    PGN_AFTERTREATMENT_2_FUEL_CONTROL_2 : UDINT := UDINT#16#FD44; (* < 64836 - AT2FC2 *)
    PGN_AFTERTREATMENT_2_THREE_WAY_CATALYST : UDINT := UDINT#16#FD45; (* < 64837 - AT2TWC *)
    PGN_AFTERTREATMENT_1_THREE_WAY_CATALYST : UDINT := UDINT#16#FD46; (* < 64838 - AT1TWC *)
    PGN_TRANSMISSION_MODE_LABELS : UDINT := UDINT#16#FD47; (* < 64839 - TML *)
    PGN_ENGINE_EXHAUST_BANK_2_O2_FUEL_TRIM : UDINT := UDINT#16#FD48; (* < 64840 - O2FT2 *)
    PGN_ENGINE_EXHAUST_BANK_1_O2_FUEL_TRIM : UDINT := UDINT#16#FD49; (* < 64841 - O2FT1 *)
    PGN_GENERAL_PURPOSE_MESSAGE_2_11 : UDINT := UDINT#16#FD4A; (* < 64842 - GPM211 *)
    PGN_GENERAL_PURPOSE_MESSAGE_2_10 : UDINT := UDINT#16#FD4B; (* < 64843 - GPM210 *)
    PGN_GENERAL_PURPOSE_MESSAGE_2_9 : UDINT := UDINT#16#FD4C; (* < 64844 - GPM29 *)
    PGN_GENERAL_PURPOSE_MESSAGE_2_8 : UDINT := UDINT#16#FD4D; (* < 64845 - GPM28 *)
    PGN_GENERAL_PURPOSE_MESSAGE_2_7 : UDINT := UDINT#16#FD4E; (* < 64846 - GPM27 *)
    PGN_GENERAL_PURPOSE_MESSAGE_2_6 : UDINT := UDINT#16#FD4F; (* < 64847 - GPM26 *)
    PGN_GENERAL_PURPOSE_MESSAGE_1_9 : UDINT := UDINT#16#FD50; (* < 64848 - GPM19 *)
    PGN_AFTERCOOLER_COOLANT_CONTROL_VALVE_COMMAND : UDINT := UDINT#16#FD51; (* < 64849 - ACCVC *)
    PGN_ENGINE_COOLANT_CONTROL_VALVE_COMMAND : UDINT := UDINT#16#FD52; (* < 64850 - ECCVC *)
    PGN_ENGINE_AVERAGE_INFORMATION : UDINT := UDINT#16#FD53; (* < 64851 - EAI *)
    PGN_DTCS_C_PREVIOUSLY_ACTIVE : UDINT := UDINT#16#FD54; (* < 64852 - DM52 *)
    PGN_DTCS_C_CONFIRMED_AND_ACTIVE : UDINT := UDINT#16#FD55; (* < 64853 - DM51 *)
    PGN_DTCS_C_PENDING : UDINT := UDINT#16#FD56; (* < 64854 - DM50 *)
    PGN_DTCS_B2_PREVIOUSLY_ACTIVE : UDINT := UDINT#16#FD57; (* < 64855 - DM49 *)
    PGN_DTCS_B2_CONFIRMED_AND_ACTIVE : UDINT := UDINT#16#FD58; (* < 64856 - DM48 *)
    PGN_DTCS_B2_PENDING : UDINT := UDINT#16#FD59; (* < 64857 - DM47 *)
    PGN_DTCS_B1_PREVIOUSLY_ACTIVE : UDINT := UDINT#16#FD5A; (* < 64858 - DM46 *)
    PGN_DTCS_B1_CONFIRMED_AND_ACTIVE : UDINT := UDINT#16#FD5B; (* < 64859 - DM45 *)
    PGN_DTCS_B1_PENDING : UDINT := UDINT#16#FD5C; (* < 64860 - DM44 *)
    PGN_DTCS_A_PREVIOUSLY_ACTIVE : UDINT := UDINT#16#FD5D; (* < 64861 - DM43 *)
    PGN_DTCS_A_CONFIRMED_AND_ACTIVE : UDINT := UDINT#16#FD5E; (* < 64862 - DM42 *)
    PGN_DTCS_A_PENDING : UDINT := UDINT#16#FD5F; (* < 64863 - DM41 *)
    PGN_HARMONIZED_B1_FAILURE_COUNTS : UDINT := UDINT#16#FD60; (* < 64864 - DM40 *)
    PGN_HARMONIZED_CUMULATIVE_CONTINUOUS_MALFUNCTION_INDICATOR_SYSTEM : UDINT := UDINT#16#FD61; (* < 64865 - DM39 *)
    PGN_HARMONIZED_GLOBAL_REGULATION_DESCRIPTION : UDINT := UDINT#16#FD62; (* < 64866 - DM38 *)
    PGN_HARMONIZED_ROADWORTHINESS_SYSTEM : UDINT := UDINT#16#FD63; (* < 64867 - DM37 *)
    PGN_HARMONIZED_ROADWORTHINESS_VEHICLE : UDINT := UDINT#16#FD64; (* < 64868 - DM36 *)
    PGN_AFTERTREATMENT_1_FUEL_CONTROL_2 : UDINT := UDINT#16#FD65; (* < 64869 - AT1FC2 *)
    PGN_ENGINE_TEMPERATURE_4 : UDINT := UDINT#16#FD66; (* < 64870 - ET4 *)
    PGN_ZERO_NET_VEHICLE_WEIGHT_CHANGE : UDINT := UDINT#16#FD67; (* < 64871 - ZNVW *)
    PGN_GROSS_COMBINATION_VEHICLE_WEIGHT : UDINT := UDINT#16#FD68; (* < 64872 - GCVW *)
    PGN_AXLE_GROUP_CALIBRATION_WEIGHTS : UDINT := UDINT#16#FD69; (* < 64873 - AGCW *)
    PGN_AXLE_GROUP_WEIGHT : UDINT := UDINT#16#FD6A; (* < 64874 - AGW *)
    PGN_AVAILABLE_AXLE_GROUP_WEIGHTS : UDINT := UDINT#16#FD6B; (* < 64875 - AAGW *)
    PGN_AFTERTREATMENT_2_AIR_CONTROL_2 : UDINT := UDINT#16#FD6C; (* < 64876 - AT2AC2 *)
    PGN_AFTERTREATMENT_1_AIR_CONTROL_2 : UDINT := UDINT#16#FD6D; (* < 64877 - AT1AC2 *)
    PGN_AFTERTREATMENT_1_SCR_SERVICE_INFORMATION_1 : UDINT := UDINT#16#FD6E; (* < 64878 - A1SCRSI1 *)
    PGN_ELECTRONIC_ENGINE_CONTROLLER_8 : UDINT := UDINT#16#FD6F; (* < 64879 - EEC8 *)
    PGN_DOOR_RAMP_CONTROL : UDINT := UDINT#16#FD70; (* < 64880 - DRC *)
    PGN_BRAKE_ACTUATOR_STROKE_STATUS : UDINT := UDINT#16#FD71; (* < 64881 - BSA *)
    PGN_ENGINE_SPARK_VOLTAGE_6 : UDINT := UDINT#16#FD72; (* < 64882 - ESV6 *)
    PGN_ENGINE_SPARK_VOLTAGE_5 : UDINT := UDINT#16#FD73; (* < 64883 - ESV5 *)
    PGN_ENGINE_SPARK_VOLTAGE_4 : UDINT := UDINT#16#FD74; (* < 64884 - ESV4 *)
    PGN_ENGINE_SPARK_VOLTAGE_3 : UDINT := UDINT#16#FD75; (* < 64885 - ESV3 *)
    PGN_ENGINE_SPARK_VOLTAGE_2 : UDINT := UDINT#16#FD76; (* < 64886 - ESV2 *)
    PGN_ENGINE_SPARK_VOLTAGE_1 : UDINT := UDINT#16#FD77; (* < 64887 - ESV1 *)
    PGN_AFTERTREATMENT_2_TRIP_INFORMATION : UDINT := UDINT#16#FD78; (* < 64888 - AT2TI *)
    PGN_AFTERTREATMENT_1_TRIP_INFORMATION : UDINT := UDINT#16#FD79; (* < 64889 - AT1TI *)
    PGN_AFTERTREATMENT_2_SERVICE_1 : UDINT := UDINT#16#FD7A; (* < 64890 - AT2S1 *)
    PGN_AFTERTREATMENT_1_SERVICE_1 : UDINT := UDINT#16#FD7B; (* < 64891 - AT1S1 *)
    PGN_DIESEL_PARTICULATE_FILTER_CONTROL_1 : UDINT := UDINT#16#FD7C; (* < 64892 - DPFC1 *)
    PGN_RESERVED_FOR_FMS_TELLTALE_STATUS : UDINT := UDINT#16#FD7D; (* < 64893 - FMS1 *)
    PGN_ADAPTIVE_FRONT_LIGHTING_SYSTEM_STATUS : UDINT := UDINT#16#FD7E; (* < 64894 - AFSS *)
    PGN_ENGINE_CONFIGURATION_2 : UDINT := UDINT#16#FD7F; (* < 64895 - EC2 *)
    PGN_EMISSION_RELATED_PERMANENT_DIAGNOSTIC_TROUBLE_CODES : UDINT := UDINT#16#FD80; (* < 64896 - DM28 *)
    PGN_EGR_COOLER_BYPASS : UDINT := UDINT#16#FD81; (* < 64897 - EGRBV *)
    PGN_ALL_PENDING_DTCS : UDINT := UDINT#16#FD82; (* < 64898 - DM27 *)
    PGN_TRANSFER_CASE_INFORMATION : UDINT := UDINT#16#FD83; (* < 64899 - TCI *)
    PGN_ENGINE_FLUID_LEVEL_PRESSURE_9 : UDINT := UDINT#16#FD84; (* < 64900 - EFL/P9 *)
    PGN_ENGINE_FLUID_LEVEL_PRESSURE_8 : UDINT := UDINT#16#FD85; (* < 64901 - EFL/P8 *)
    PGN_ENGINE_FLUID_LEVEL_PRESSURE_7 : UDINT := UDINT#16#FD86; (* < 64902 - EFL/P7 *)
    PGN_ENGINE_FLUID_LEVEL_PRESSURE_6 : UDINT := UDINT#16#FD87; (* < 64903 - EFL/P6 *)
    PGN_ENGINE_FLUID_LEVEL_PRESSURE_5 : UDINT := UDINT#16#FD88; (* < 64904 - EFL/P5 *)
    PGN_VEHICLE_DIRECTION_SPEED_2 : UDINT := UDINT#16#FD89; (* < 64905 - VDS2 *)
    PGN_SAE_J2012_2_BYTE_DTC_DISPLAY : UDINT := UDINT#16#FD8A; (* < 64906 - J2012_2B *)
    PGN_AFTERTREATMENT_2_GAS_PARAMETERS : UDINT := UDINT#16#FD8B; (* < 64907 - AT2GP *)
    PGN_AFTERTREATMENT_1_GAS_PARAMETERS : UDINT := UDINT#16#FD8C; (* < 64908 - AT1GP *)
    PGN_UTILITY_TOTAL_AC_REACTIVE_ENERGY : UDINT := UDINT#16#FD8D; (* < 64909 - UTACER *)
    PGN_GENERATOR_TOTAL_AC_REACTIVE_ENERGY : UDINT := UDINT#16#FD8E; (* < 64910 - GTACER *)
    PGN_GENERATOR_TOTAL_AC_PERCENT_POWER : UDINT := UDINT#16#FD8F; (* < 64911 - GTACPP *)
    PGN_ADVERTISED_ENGINE_TORQUE_CURVE : UDINT := UDINT#16#FD90; (* < 64912 - AETC *)
    PGN_AC_SWITCHING_DEVICE_STATUS : UDINT := UDINT#16#FD91; (* < 64913 - ACS *)
    PGN_ENGINE_OPERATING_INFORMATIO : UDINT := UDINT#16#FD92; (* < 64914 - EOI *)
    PGN_GENERATOR_CONTROL_1 : UDINT := UDINT#16#FD93; (* < 64915 - GC1 *)
    PGN_ELECTRONIC_ENGINE_CONTROLLER_7 : UDINT := UDINT#16#FD94; (* < 64916 - EEC7 *)
    PGN_TRANSMISSION_FLUIDS_2 : UDINT := UDINT#16#FD95; (* < 64917 - TRF2 *)
    PGN_FUEL_INFORMATION_2_LIQUID : UDINT := UDINT#16#FD96; (* < 64918 - LFI2 *)
    PGN_FUEL_INFORMATION_3_LIQUID : UDINT := UDINT#16#FD97; (* < 64919 - LFI3 *)
    PGN_AFTERTREATMENT_1_HISTORICAL_INFORMATION_1 : UDINT := UDINT#16#FD98; (* < 64920 - AT1HI1 *)
    PGN_AFTERTREATMENT_2_HISTORICAL_INFORMATION_1 : UDINT := UDINT#16#FD99; (* < 64921 - AT2HI1 *)
    PGN_ELECTRONIC_BRAKE_SYSTEM_2_4 : UDINT := UDINT#16#FD9A; (* < 64922 - EBS24 *)
    PGN_AFTERTREATMENT_1_DIESEL_EXHAUST_FLUID_INFORMATION_1 : UDINT := UDINT#16#FD9B; (* < 64923 - A1DEFI1 *)
    PGN_SENSOR_ELECTRICAL_POWER_2 : UDINT := UDINT#16#FD9C; (* < 64924 - SEP2 *)
    PGN_SENSOR_ELECTRICAL_POWER_1 : UDINT := UDINT#16#FD9D; (* < 64925 - SEP1 *)
    PGN_AFTERTREATMENT_2_AIR_CONTROL_1 : UDINT := UDINT#16#FD9E; (* < 64926 - AT2AC1 *)
    PGN_AFTERTREATMENT_1_AIR_CONTROL_1 : UDINT := UDINT#16#FD9F; (* < 64927 - AT1AC1 *)
    PGN_AFTERTREATMENT_2_FUEL_CONTROL_1 : UDINT := UDINT#16#FDA0; (* < 64928 - AT2FC1 *)
    PGN_AFTERTREATMENT_1_FUEL_CONTROL_1 : UDINT := UDINT#16#FDA1; (* < 64929 - AT1FC1 *)
    PGN_FUEL_INFORMATION_3_GASEOUS : UDINT := UDINT#16#FDA2; (* < 64930 - GFI3 *)
    PGN_ELECTRONIC_ENGINE_CONTROLLER_6 : UDINT := UDINT#16#FDA3; (* < 64931 - EEC6 *)
    PGN_PTO_DRIVE_ENGAGEMENT_1 : UDINT := UDINT#16#FDA4; (* < 64932 - PTODE1 *)
    PGN_DOOR_CONTROL_2 : UDINT := UDINT#16#FDA5; (* < 64933 - DC2 *)
    PGN_VOLTAGE_REGULATOR_EXCITATION_STATUS : UDINT := UDINT#16#FDA6; (* < 64934 - VREP *)
    PGN_VOLTAGE_REGULATOR_OPERATING_MODE : UDINT := UDINT#16#FDA7; (* < 64935 - VROM *)
    PGN_WIRELESS_COMMUNICATIONS_MESSAGE_2 : UDINT := UDINT#16#FDA8; (* < 64936 - WCM2 *)
    PGN_WCM1 : UDINT := UDINT#16#FDA9; (* < 64937 - WCM1 *)
    PGN_ENGINE_FLUID_LEVEL_PRESSURE_4 : UDINT := UDINT#16#FDAA; (* < 64938 - EFL/P4 *)
    PGN_REQUEST_FOR_COMPLETE_CONFIGURABLE_MESSAGE_SET_NO_LONGER_USED : UDINT := UDINT#16#FDAB; (* < 64939 - Request For Complete Configurable Message Set (no longer used) *)
    PGN_ENGINE_FUEL_INFORMATION : UDINT := UDINT#16#FDAC; (* < 64940 - EFI *)
    PGN_REQUEST_FOR_COMPLETE_CONFIGURABLE_MESSAGE_SET : UDINT := UDINT#16#FDAD; (* < 64941 - RCMS *)
    PGN_FIFTH_WHEEL_SMART_SYSTEMS_2 : UDINT := UDINT#16#FDAE; (* < 64942 - FWSS2 *)
    PGN_AFTERTREATMENT_2_INTERMEDIATE_GAS : UDINT := UDINT#16#FDAF; (* < 64943 - AT2IMG *)
    PGN_AFTERTREATMENT_2_OUTLET_GAS_2 : UDINT := UDINT#16#FDB0; (* < 64944 - AT2OG2 *)
    PGN_AFTERTREATMENT_2_INTAKE_GAS_2 : UDINT := UDINT#16#FDB1; (* < 64945 - AT2IG2 *)
    PGN_AFTERTREATMENT_1_INTERMEDIATE_GAS : UDINT := UDINT#16#FDB2; (* < 64946 - AT1IMG *)
    PGN_AFTERTREATMENT_1_OUTLET_GAS_2 : UDINT := UDINT#16#FDB3; (* < 64947 - AT1OG2 *)
    PGN_AFTERTREATMENT_1_INTAKE_GAS_2 : UDINT := UDINT#16#FDB4; (* < 64948 - AT1IG2 *)
    PGN_EMISSION_RELATED_PREVIOUSLY_MIL_ON_DIAGNOSTIC_TROUBLE_CODES : UDINT := UDINT#16#FDB5; (* < 64949 - DM23 *)
    PGN_SPN_SUPPORT : UDINT := UDINT#16#FDB6; (* < 64950 - DM24 *)
    PGN_EXPANDED_FREEZE_FRAME : UDINT := UDINT#16#FDB7; (* < 64951 - DM25 *)
    PGN_DIAGNOSTIC_READINESS_3 : UDINT := UDINT#16#FDB8; (* < 64952 - DM26 *)
    PGN_TIRE_PRESSURE_REFERENCE_INFORMATION : UDINT := UDINT#16#FDB9; (* < 64953 - TPRI *)
    PGN_FAREBOX_STATUS : UDINT := UDINT#16#FDBA; (* < 64954 - TR6 *)
    PGN_FAREBOX_POINT_OF_SALE : UDINT := UDINT#16#FDBB; (* < 64955 - TR5 *)
    PGN_FAREBOX_SERVICE_DETAIL : UDINT := UDINT#16#FDBC; (* < 64956 - TR4 *)
    PGN_SIGNAL_PREEMPTION : UDINT := UDINT#16#FDBD; (* < 64957 - TR3 *)
    PGN_TRANSIT_ROUTE : UDINT := UDINT#16#FDBE; (* < 64958 - TR1 *)
    PGN_TRANSIT_MILEPOST : UDINT := UDINT#16#FDBF; (* < 64959 - TR2 *)
    PGN_PASSENGER_COUNTER : UDINT := UDINT#16#FDC0; (* < 64960 - TR7 *)
    PGN_ENGINE_FLUID_LEVEL_PRESSURE_3 : UDINT := UDINT#16#FDC1; (* < 64961 - EFL/P3 *)
    PGN_ELECTRONIC_ENGINE_CONTROLLER_14 : UDINT := UDINT#16#FDC2; (* < 64962 - EEC14 *)
    PGN_ELECTRONIC_ENGINE_CONTROLLER_15 : UDINT := UDINT#16#FDC3; (* < 64963 - EEC15 *)
    PGN_ELECTRONIC_BRAKE_CONTROLLER_5 : UDINT := UDINT#16#FDC4; (* < 64964 - EBC5 *)
    PGN_ECU_IDENTIFICATION_INFO : UDINT := UDINT#16#FDC5; (* < 64965 - ECUID *)
    PGN_COLD_START_AIDS : UDINT := UDINT#16#FDC6; (* < 64966 - CSA *)
    PGN_OFF_HIGHWAY_ENGINE_CONTROL_SELECTION_STATES : UDINT := UDINT#16#FDC7; (* < 64967 - OHCSS *)
    PGN_OPERATOR_PRIMARY_INTERMEDIATE_SPEED_CONTROL_STATE : UDINT := UDINT#16#FDC8; (* < 64968 - ISCS *)
    PGN_ELECTRONIC_CONTROL_MODULE_INFORMATION : UDINT := UDINT#16#FDC9; (* < 64969 - CMI *)
    PGN_INTERMEDIATE_SPEED_CONTROL : UDINT := UDINT#16#FDCA; (* < 64970 - ISC *)
    PGN_OFFHIGHW_ENGINE_CTRL_SELECT : UDINT := UDINT#16#FDCB; (* < 64971 - OHECS *)
    PGN_OPERATORS_EXTERNAL_LIGHT_CONTROLS_MESSAGE : UDINT := UDINT#16#FDCC; (* < 64972 - OEL *)
    PGN_OPERATOR_WIPER_AND_WASHER_CONTROLS_MESSAGE : UDINT := UDINT#16#FDCD; (* < 64973 - OWW *)
    PGN_WORKING_SET_MEMBER_MESSAGE_OBSOLETE_SEE_PGN_65088 : UDINT := UDINT#16#FDCE; (* < 64974 - WSMM *)
    PGN_WORKING_SET_MASTER_MESSAGE_OBSOLETE_SEE_PGN_65089 : UDINT := UDINT#16#FDCF; (* < 64975 - WSM *)
    PGN_INTAKE_EXHAUST_CONDITIONS_2 : UDINT := UDINT#16#FDD0; (* < 64976 - IC2 *)
    PGN_FMS_STANDARD_INTERFAC_IDENT : UDINT := UDINT#16#FDD1; (* < 64977 - FMS *)
    PGN_ECU_PERFORMANCE : UDINT := UDINT#16#FDD2; (* < 64978 - EP *)
    PGN_TURBOCHARGER_INFORMATION_6 : UDINT := UDINT#16#FDD3; (* < 64979 - TCI6 *)
    PGN_CAB_MESSAGE_3 : UDINT := UDINT#16#FDD4; (* < 64980 - CM3 *)
    PGN_ELEC_ENGINE_CONTROLLER_5 : UDINT := UDINT#16#FDD5; (* < 64981 - EEC5 *)
    PGN_BASIC_JOYSTICK_MESSAGE_1 : UDINT := UDINT#16#FDD6; (* < 64982 - BJM1 *)
    PGN_EXTENDED_JOYSTICK_MESSAGE_1 : UDINT := UDINT#16#FDD7; (* < 64983 - EJM1 *)
    PGN_BASIC_JOYSTICK_MESSAGE_2 : UDINT := UDINT#16#FDD8; (* < 64984 - BJM2 *)
    PGN_EXTENDED_JOYSTICK_MESSAGE_2 : UDINT := UDINT#16#FDD9; (* < 64985 - EJM2 *)
    PGN_BASIC_JOYSTICK_MESSAGE_3 : UDINT := UDINT#16#FDDA; (* < 64986 - BJM3 *)
    PGN_EXTENDED_JOYSTICK_MESSAGE_3 : UDINT := UDINT#16#FDDB; (* < 64987 - EJM3 *)
    PGN_MARINE_CONTROL_INFORMATION : UDINT := UDINT#16#FDDC; (* < 64988 - MCI *)
    PGN_MILITARY_APPLICATION_MESSAGE_1_1 : UDINT := UDINT#16#FDDD; (* < 64989 - MAM11 *)
    PGN_AMBIENT_CONDITIONS_2 : UDINT := UDINT#16#FDDE; (* < 64990 - MAM21 *)
    PGN_FRONT_WHEEL_DRIVE_STATUS : UDINT := UDINT#16#FDDF; (* < 64991 - FWD *)
    PGN_AMBIENT_CONDITIONS_2_64992 : UDINT := UDINT#16#FDE0; (* < 64992 - AMB2 *)
    PGN_CAB_A_C_CLIMATE_SYST_INFO : UDINT := UDINT#16#FDE1; (* < 64993 - CCSI1 *)
    PGN_SUPPLY_PRESSURE_DEMAND : UDINT := UDINT#16#FDE2; (* < 64994 - SPR *)
    PGN_EQUIPM_OPERATION_AND_CONTR : UDINT := UDINT#16#FDE3; (* < 64995 - EOAC *)
    PGN_EQUIPMENT_PERFORMANCE_DATA : UDINT := UDINT#16#FDE4; (* < 64996 - EPD *)
    PGN_MAX_VEHIC_SPEED_LIMIT_STAT : UDINT := UDINT#16#FDE5; (* < 64997 - MVS *)
    PGN_HYDRAULIC_BRAKING_SYSTEM : UDINT := UDINT#16#FDE6; (* < 64998 - HBS *)
    PGN_BUS_1_UTIL_SYNC_CHECK_STATU : UDINT := UDINT#16#FDE7; (* < 64999 - BUSC *)
    PGN_BUS_1_GENERA_SYNC_CH_STAT : UDINT := UDINT#16#FDE8; (* < 65000 - BGSC *)
    PGN_BUS_1_PHASE_C_BASIC_AC_QUAN : UDINT := UDINT#16#FDE9; (* < 65001 - BPCAC *)
    PGN_BUS_1_PHASE_B_BASIC_AC_QUAN : UDINT := UDINT#16#FDEA; (* < 65002 - BPBAC *)
    PGN_BUS_1_PHASE_A_BASIC_AC_QUAN : UDINT := UDINT#16#FDEB; (* < 65003 - BPAAC *)
    PGN_BUS_1_AVERAGE_BASIC_AC_QUAN : UDINT := UDINT#16#FDEC; (* < 65004 - BAAC *)
    PGN_UTIL_TOTAL_AC_ENERGY : UDINT := UDINT#16#FDED; (* < 65005 - UTACE *)
    PGN_UTIL_PHASE_C_AC_REACT_POWER : UDINT := UDINT#16#FDEE; (* < 65006 - UPCACR *)
    PGN_UTIL_PHASE_C_AC_POWER : UDINT := UDINT#16#FDEF; (* < 65007 - UPCACP *)
    PGN_UTIL_PHASE_C_AC_BASIC_QUANT : UDINT := UDINT#16#FDF0; (* < 65008 - UPCAC *)
    PGN_UTIL_PHASE_B_AC_REACT_POWER : UDINT := UDINT#16#FDF1; (* < 65009 - UPBACR *)
    PGN_UTIL_PHASE_B_AC_POWER : UDINT := UDINT#16#FDF2; (* < 65010 - UPBACP *)
    PGN_UTIL_PHASE_B_AC_BASIC_QUANT : UDINT := UDINT#16#FDF3; (* < 65011 - UPBAC *)
    PGN_UTIL_PHASE_A_AC_REACT_POWER : UDINT := UDINT#16#FDF4; (* < 65012 - UPACCR *)
    PGN_UTIL_PHASE_A_AC_POWER : UDINT := UDINT#16#FDF5; (* < 65013 - UPAACP *)
    PGN_UTIL_PHASE_A_AC_BASIC_QUANT : UDINT := UDINT#16#FDF6; (* < 65014 - UPAAC *)
    PGN_UTIL_AC_REACTIVE_POWER : UDINT := UDINT#16#FDF7; (* < 65015 - UTACR *)
    PGN_UTIL_TOTAL_AC_POWER : UDINT := UDINT#16#FDF8; (* < 65016 - UTACP *)
    PGN_UTIL_AVERACE_BASIC_AC_QUANT : UDINT := UDINT#16#FDF9; (* < 65017 - UAAC *)
    PGN_GENERATOR_TOTAL_AC_ENERGY : UDINT := UDINT#16#FDFA; (* < 65018 - GTACE *)
    PGN_GENERA_PHAS_C_AC_REACT_PWR : UDINT := UDINT#16#FDFB; (* < 65019 - GPCACR *)
    PGN_GENERATOR_PHASE_C_AC_POWER : UDINT := UDINT#16#FDFC; (* < 65020 - GPCACP *)
    PGN_GENERA_PHASE_C_BAS_AC_QUANT : UDINT := UDINT#16#FDFD; (* < 65021 - GPCAC *)
    PGN_GENERA_PHASE_B_AC_REACT_PWR : UDINT := UDINT#16#FDFE; (* < 65022 - GPBACRP *)
    PGN_GENERATOR_PHASE_B_AC_POWER : UDINT := UDINT#16#FDFF; (* < 65023 - GPBACP *)
    PGN_PDU2_254_Y : UDINT := UDINT#16#FE00; (* < 65024 - GPBAC *)
    PGN_GENERA_PHASE_B_BAS_AC_QUANT : UDINT := UDINT#16#FE00; (* < 65024 - GPBAC *)
    PGN_GENERA_PHASE_A_AC_REACT_PWR : UDINT := UDINT#16#FE01; (* < 65025 - GPAACR *)
    PGN_GENERATOR_PHASE_A_AC_POWER : UDINT := UDINT#16#FE02; (* < 65026 - GPAACP *)
    PGN_GENERA_PHASE_A_BAS_AC_QUANT : UDINT := UDINT#16#FE03; (* < 65027 - GPAAC *)
    PGN_GENERA_TOTAL_AC_REACT_POWER : UDINT := UDINT#16#FE04; (* < 65028 - GTACR *)
    PGN_GENERATOR_TOTAL_AC_POWER : UDINT := UDINT#16#FE05; (* < 65029 - GTACP *)
    PGN_GENERA_TOTAL_BAS_AC_QUANTI : UDINT := UDINT#16#FE06; (* < 65030 - GAAC *)
    PGN_EXHAUST_TEMPERATURE : UDINT := UDINT#16#FE07; (* < 65031 - ET *)
    PGN_REQUIRED_TRACTOR_FACILITIES : UDINT := UDINT#16#FE08; (* < 65032 - RTF *)
    PGN_TRACTOR_FACILITIES_RESPONSE : UDINT := UDINT#16#FE09; (* < 65033 - TFR *)
    PGN_IMP_REMOTE_CMD_TRACTOR_RESP : UDINT := UDINT#16#FE0A; (* < 65034 - IRCR *)
    PGN_IMPLEMENT_REMOTE_CONTR_CMD : UDINT := UDINT#16#FE0B; (* < 65035 - IRC *)
    PGN_WORKING_SET_MEMBER : UDINT := UDINT#16#FE0C; (* < 65036 - WSMEM *)
    PGN_WORKING_SET_MASTER : UDINT := UDINT#16#FE0D; (* < 65037 - WSMSTR *)
    PGN_RESP_FOR_REPETITION_RATE : UDINT := UDINT#16#FE0E; (* < 65038 - RESRR *)
    PGN_LANGUAGE_COMMAND : UDINT := UDINT#16#FE0F; (* < 65039 - LC *)
    PGN_AUX_VALVE_0_EST_FLOW : UDINT := UDINT#16#FE10; (* < 65040 - AV00EF *)
    PGN_AUX_VALVE_1_EST_FLOW : UDINT := UDINT#16#FE11; (* < 65041 - AV01EF *)
    PGN_AUX_VALVE_2_EST_FLOW : UDINT := UDINT#16#FE12; (* < 65042 - AV02EF *)
    PGN_AUX_VALVE_3_EST_FLOW : UDINT := UDINT#16#FE13; (* < 65043 - AV03EF *)
    PGN_AUX_VALVE_4_EST_FLOW : UDINT := UDINT#16#FE14; (* < 65044 - AV04EF *)
    PGN_AUX_VALVE_5_EST_FLOW : UDINT := UDINT#16#FE15; (* < 65045 - AV05EF *)
    PGN_AUX_VALVE_6_EST_FLOW : UDINT := UDINT#16#FE16; (* < 65046 - AV06EF *)
    PGN_AUX_VALVE_7_EST_FLOW : UDINT := UDINT#16#FE17; (* < 65047 - AV07EF *)
    PGN_AUX_VALVE_8_EST_FLOW : UDINT := UDINT#16#FE18; (* < 65048 - AV08EF *)
    PGN_AUX_VALVE_9_EST_FLOW : UDINT := UDINT#16#FE19; (* < 65049 - AV09EF *)
    PGN_AUX_VALVE_10_EST_FLOW : UDINT := UDINT#16#FE1A; (* < 65050 - AV10EF *)
    PGN_AUX_VALVE_11_EST_FLOW : UDINT := UDINT#16#FE1B; (* < 65051 - AV11EF *)
    PGN_AUX_VALVE_12_EST_FLOW : UDINT := UDINT#16#FE1C; (* < 65052 - AV12EF *)
    PGN_AUX_VALVE_13_EST_FLOW : UDINT := UDINT#16#FE1D; (* < 65053 - AV13EF *)
    PGN_AUX_VALVE_14_EST_FLOW : UDINT := UDINT#16#FE1E; (* < 65054 - AV14EF *)
    PGN_AUX_VALVE_15_EST_FLOW : UDINT := UDINT#16#FE1F; (* < 65055 - AV15EF *)
    PGN_AUX_VALVE_0_MEAS_FLOW : UDINT := UDINT#16#FE20; (* < 65056 - AV00MF *)
    PGN_AUX_VALVE_1_MEAS_FLOW : UDINT := UDINT#16#FE21; (* < 65057 - AV01MF *)
    PGN_AUX_VALVE_2_MEAS_FLOW : UDINT := UDINT#16#FE22; (* < 65058 - AV02MF *)
    PGN_AUX_VALVE_3_MEAS_FLOW : UDINT := UDINT#16#FE23; (* < 65059 - AV03MF *)
    PGN_AUX_VALVE_4_MEAS_FLOW : UDINT := UDINT#16#FE24; (* < 65060 - AV04MF *)
    PGN_AUX_VALVE_5_MEAS_FLOW : UDINT := UDINT#16#FE25; (* < 65061 - AV05MF *)
    PGN_AUX_VALVE_6_MEAS_FLOW : UDINT := UDINT#16#FE26; (* < 65062 - AV06MF *)
    PGN_AUX_VALVE_7_MEAS_FLOW : UDINT := UDINT#16#FE27; (* < 65063 - AV07MF *)
    PGN_AUX_VALVE_8_MEAS_FLOW : UDINT := UDINT#16#FE28; (* < 65064 - AV08MF *)
    PGN_AUX_VALVE_9_MEAS_FLOW : UDINT := UDINT#16#FE29; (* < 65065 - AV09MF *)
    PGN_AUX_VALVE_10_MEAS_FLOW : UDINT := UDINT#16#FE2A; (* < 65066 - AV10MF *)
    PGN_AUX_VALVE_11_MEAS_FLOW : UDINT := UDINT#16#FE2B; (* < 65067 - AV11MF *)
    PGN_AUX_VALVE_12_MEAS_FLOW : UDINT := UDINT#16#FE2C; (* < 65068 - AV12MF *)
    PGN_AUX_VALVE_13_MEAS_FLOW : UDINT := UDINT#16#FE2D; (* < 65069 - AV13MF *)
    PGN_AUX_VALVE_14_MEAS_FLOW : UDINT := UDINT#16#FE2E; (* < 65070 - AV14MF *)
    PGN_AUX_VALVE_15_MEAS_FLOW : UDINT := UDINT#16#FE2F; (* < 65071 - AV15MF *)
    PGN_AUX_VALVE_0_COMMAND : UDINT := UDINT#16#FE30; (* < 65072 - AV00C *)
    PGN_AUX_VALVE_1_COMMAND : UDINT := UDINT#16#FE31; (* < 65073 - AV01C *)
    PGN_AUX_VALVE_2_COMMAND : UDINT := UDINT#16#FE32; (* < 65074 - AV02C *)
    PGN_AUX_VALVE_3_COMMAND : UDINT := UDINT#16#FE33; (* < 65075 - AV03C *)
    PGN_AUX_VALVE_4_COMMAND : UDINT := UDINT#16#FE34; (* < 65076 - AV04C *)
    PGN_AUX_VALVE_5_COMMAND : UDINT := UDINT#16#FE35; (* < 65077 - AV05C *)
    PGN_AUX_VALVE_6_COMMAND : UDINT := UDINT#16#FE36; (* < 65078 - AV06C *)
    PGN_AUX_VALVE_7_COMMAND : UDINT := UDINT#16#FE37; (* < 65079 - AV07C *)
    PGN_AUX_VALVE_8_COMMAND : UDINT := UDINT#16#FE38; (* < 65080 - AV08C *)
    PGN_AUX_VALVE_9_COMMAND : UDINT := UDINT#16#FE39; (* < 65081 - AV09C *)
    PGN_AUX_VALVE_10_COMMAND : UDINT := UDINT#16#FE3A; (* < 65082 - AV10C *)
    PGN_AUX_VALVE_11_COMMAND : UDINT := UDINT#16#FE3B; (* < 65083 - AV11C *)
    PGN_AUX_VALVE_12_COMMAND : UDINT := UDINT#16#FE3C; (* < 65084 - AV12C *)
    PGN_AUX_VALVE_13_COMMAND : UDINT := UDINT#16#FE3D; (* < 65085 - AV13C *)
    PGN_AUX_VALVE_14_COMMAND : UDINT := UDINT#16#FE3E; (* < 65086 - AV14C *)
    PGN_AUX_VALVE_15_COMMAND : UDINT := UDINT#16#FE3F; (* < 65087 - AV15C *)
    PGN_LIGHTING_DATA : UDINT := UDINT#16#FE40; (* < 65088 - LD *)
    PGN_LIGHTING_COMMAND : UDINT := UDINT#16#FE41; (* < 65089 - LCMD *)
    PGN_COMMAND_HITCH_PTO : UDINT := UDINT#16#FE42; (* < 65090 - HPTOC *)
    PGN_REAR_PTO : UDINT := UDINT#16#FE43; (* < 65091 - RPTO *)
    PGN_FRONT_PTO : UDINT := UDINT#16#FE44; (* < 65092 - FPTO *)
    PGN_REAR_HITCH : UDINT := UDINT#16#FE45; (* < 65093 - RHS *)
    PGN_FRONT_HITCH : UDINT := UDINT#16#FE46; (* < 65094 - FHS *)
    PGN_MAINTAIN_POWER : UDINT := UDINT#16#FE47; (* < 65095 - MP *)
    PGN_WHEEL_BASED_SPEED : UDINT := UDINT#16#FE48; (* < 65096 - WBSD *)
    PGN_GROUND_BASED_SPEED : UDINT := UDINT#16#FE49; (* < 65097 - GBSD *)
    PGN_ELECTRONIC_TRANSMISSION_CONTROLLER_7 : UDINT := UDINT#16#FE4A; (* < 65098 - ETC7 *)
    PGN_TRANSMISSIONG_CONFIG_2 : UDINT := UDINT#16#FE4B; (* < 65099 - TCFG2 *)
    PGN_MILITARY_LIGHTING_COMMAND : UDINT := UDINT#16#FE4C; (* < 65100 - ML *)
    PGN_TOTAL_AVERAGED_INFORMATION : UDINT := UDINT#16#FE4D; (* < 65101 - TAVG *)
    PGN_DOOR_CONTROL : UDINT := UDINT#16#FE4E; (* < 65102 - DC1 *)
    PGN_VEHICLE_DYN_STAB_CTRL_1 : UDINT := UDINT#16#FE4F; (* < 65103 - VDC1 *)
    PGN_BATTERY_TEMPERATURE : UDINT := UDINT#16#FE50; (* < 65104 - BT1 *)
    PGN_ADAPT_CRUISE_CONTR_OPER_INP : UDINT := UDINT#16#FE51; (* < 65105 - ACC2 *)
    PGN_VEHICLE_ELECTRICAL_POWER_3 : UDINT := UDINT#16#FE52; (* < 65106 - VEP3 *)
    PGN_RETARD_TORQUE_SPEED_LIMIT : UDINT := UDINT#16#FE53; (* < 65107 - RTC1 *)
    PGN_ENGINE_TORQUE_SPEED_LIMIT : UDINT := UDINT#16#FE54; (* < 65108 - ECT1 *)
    PGN_GASEOUS_FUEL_PROPERTIES : UDINT := UDINT#16#FE55; (* < 65109 - GFD *)
    PGN_TANK_INFORMATION_1 : UDINT := UDINT#16#FE56; (* < 65110 - AT1T1I1 *)
    PGN_AIR_SUSPENSION_CONTROL_5 : UDINT := UDINT#16#FE57; (* < 65111 - ASC5 *)
    PGN_AIR_SUSPENSION_CONTROL_4 : UDINT := UDINT#16#FE58; (* < 65112 - ASC4 *)
    PGN_AIR_SUSPENSION_CONTROL_3 : UDINT := UDINT#16#FE59; (* < 65113 - ASC3 *)
    PGN_AIR_SUSPENSION_CONTROL_1 : UDINT := UDINT#16#FE5A; (* < 65114 - ASC1 *)
    PGN_FORWARD_LANE_IMAGE : UDINT := UDINT#16#FE5B; (* < 65115 - FLI2 *)
    PGN_RUNNING_GEAR_EQUIPMENT_2_2 : UDINT := UDINT#16#FE5C; (* < 65116 - RGE22 *)
    PGN_GENERAL_PURPOSE_MESSAGE_1_2 : UDINT := UDINT#16#FE5D; (* < 65117 - GPM12 *)
    PGN_RUNNING_GEAR_EQUIPMENT_2_3 : UDINT := UDINT#16#FE5E; (* < 65118 - RGE23 *)
    PGN_GENERAL_PURPOSE_MESSAGE_1_3 : UDINT := UDINT#16#FE5F; (* < 65119 - GPM13 *)
    PGN_GENERAL_PURPOSE_MESSAGE_2_3 : UDINT := UDINT#16#FE60; (* < 65120 - GPM23 *)
    PGN_GENERAL_PURPOSE_MESSAGE_1_4 : UDINT := UDINT#16#FE61; (* < 65121 - GPM14 *)
    PGN_GENERAL_PURPOSE_MESSAGE_2_4 : UDINT := UDINT#16#FE62; (* < 65122 - GPM24 *)
    PGN_GENERAL_PURPOSE_MESSAGE_1_5 : UDINT := UDINT#16#FE63; (* < 65123 - GPM15 *)
    PGN_GENERAL_PURPOSE_MESSAGE_2_5 : UDINT := UDINT#16#FE64; (* < 65124 - GPM25 *)
    PGN_GENERAL_PURPOSE_MESSAGE_1_6 : UDINT := UDINT#16#FE65; (* < 65125 - GPM16 *)
    PGN_BATTERY_MAIN_SWITCH_INFO : UDINT := UDINT#16#FE66; (* < 65126 - BM *)
    PGN_CLIMATE_CONTR_CONFIGURATION : UDINT := UDINT#16#FE67; (* < 65127 - CCC *)
    PGN_VEHICLE_FLUIDS : UDINT := UDINT#16#FE68; (* < 65128 - VF *)
    PGN_ENGINE_TEMPERATURE_3 : UDINT := UDINT#16#FE69; (* < 65129 - ET3 *)
    PGN_ENGINE_FUEL_LUBE_SYSTEMS : UDINT := UDINT#16#FE6A; (* < 65130 - EFS *)
    PGN_DRIVERS_IDENTIFICATION : UDINT := UDINT#16#FE6B; (* < 65131 - DI *)
    PGN_TACHOGRAPH : UDINT := UDINT#16#FE6C; (* < 65132 - TCO1 *)
    PGN_HEATER_INFORMATION : UDINT := UDINT#16#FE6D; (* < 65133 - HTR *)
    PGN_HIGH_RESOLUTION_WHEEL_SPEED : UDINT := UDINT#16#FE6E; (* < 65134 - HRW *)
    PGN_ADAPTIVE_CRUISE_CONTROL : UDINT := UDINT#16#FE6F; (* < 65135 - ACC1 *)
    PGN_COMBINATION_VEHICLE_WEIGHT : UDINT := UDINT#16#FE70; (* < 65136 - CVW *)
    PGN_LASER_TRACER_POSITION : UDINT := UDINT#16#FE71; (* < 65137 - LTP *)
    PGN_LASER_LEVEL_SYS_BLADE_CONTR : UDINT := UDINT#16#FE72; (* < 65138 - LBC *)
    PGN_LASER_RECEIVER_MAST_POS : UDINT := UDINT#16#FE73; (* < 65139 - LMP *)
    PGN_MODIFY_LEVEL_CTRL_SET_POINT : UDINT := UDINT#16#FE74; (* < 65140 - LSP *)
    PGN_LASER_LVL_SYS_VERTIC_DEVIAT : UDINT := UDINT#16#FE75; (* < 65141 - LVD *)
    PGN_LASER_LVL_SYS_POS_DISP_DATA : UDINT := UDINT#16#FE76; (* < 65142 - LVDD *)
    PGN_AUXILIARY_PRESSURES : UDINT := UDINT#16#FE77; (* < 65143 - AP *)
    PGN_TIRE_PRESS_CONTR_UNIT_STAT : UDINT := UDINT#16#FE78; (* < 65144 - TP1 *)
    PGN_TIRE_PRESS_CTRL_TARGET_PRES : UDINT := UDINT#16#FE79; (* < 65145 - TP2 *)
    PGN_TIRE_PRESS_UNIT_CURR_PRESS : UDINT := UDINT#16#FE7A; (* < 65146 - TP3 *)
    PGN_COMBUSTION_TIME_1 : UDINT := UDINT#16#FE7B; (* < 65147 - CT1 *)
    PGN_COMBUSTION_TIME_2 : UDINT := UDINT#16#FE7C; (* < 65148 - CT2 *)
    PGN_COMBUSTION_TIME_3 : UDINT := UDINT#16#FE7D; (* < 65149 - CT3 *)
    PGN_COMBUSTION_TIME_4 : UDINT := UDINT#16#FE7E; (* < 65150 - CT4 *)
    PGN_COMBUSTION_TIME_5 : UDINT := UDINT#16#FE7F; (* < 65151 - CT5 *)
    PGN_COMBUSTION_TIME_6 : UDINT := UDINT#16#FE80; (* < 65152 - CT6 *)
    PGN_FUEL_INFORMATION_2 : UDINT := UDINT#16#FE81; (* < 65153 - GFI2 *)
    PGN_IGNITION_TIMING_1 : UDINT := UDINT#16#FE82; (* < 65154 - IT1 *)
    PGN_IGNITION_TIMING_2 : UDINT := UDINT#16#FE83; (* < 65155 - IT2 *)
    PGN_IGNITION_TIMING_3 : UDINT := UDINT#16#FE84; (* < 65156 - IT3 *)
    PGN_IGNITION_TIMING_4 : UDINT := UDINT#16#FE85; (* < 65157 - IT4 *)
    PGN_IGNITION_TIMING_5 : UDINT := UDINT#16#FE86; (* < 65158 - IT5 *)
    PGN_IGNITION_TIMING_6 : UDINT := UDINT#16#FE87; (* < 65159 - IT6 *)
    PGN_IGNITION_TRANSF_SECOND_OP1 : UDINT := UDINT#16#FE88; (* < 65160 - ISO1 *)
    PGN_IGNITION_TRANSF_SECOND_OP2 : UDINT := UDINT#16#FE89; (* < 65161 - ISO2 *)
    PGN_IGNITION_TRANSF_SECOND_OP3 : UDINT := UDINT#16#FE8A; (* < 65162 - ISO3 *)
    PGN_GASEOUS_FUEL_PRESSURE : UDINT := UDINT#16#FE8B; (* < 65163 - GFP1 *)
    PGN_AUXILIARY_ANALOG_INFO : UDINT := UDINT#16#FE8C; (* < 65164 - AAI *)
    PGN_VEHICLE_ELECTRICAL_POWER_2 : UDINT := UDINT#16#FE8D; (* < 65165 - VEP2 *)
    PGN_SERVICE_2 : UDINT := UDINT#16#FE8E; (* < 65166 - S2 *)
    PGN_SUPPLY_PRESSURE_2 : UDINT := UDINT#16#FE8F; (* < 65167 - SP2 *)
    PGN_ENGINE_TORQUE_HISTORY : UDINT := UDINT#16#FE90; (* < 65168 - ETH *)
    PGN_FUEL_LEAKAGE : UDINT := UDINT#16#FE91; (* < 65169 - FL *)
    PGN_ENGINE_INFORMATION : UDINT := UDINT#16#FE92; (* < 65170 - EI1 *)
    PGN_ENGINE_ELECTR_SYST_MOD_INFO : UDINT := UDINT#16#FE93; (* < 65171 - EES *)
    PGN_ENGINE_AUXILIARY_COOLANT : UDINT := UDINT#16#FE94; (* < 65172 - EAC *)
    PGN_REBUILD_INFORMATION : UDINT := UDINT#16#FE95; (* < 65173 - RBI *)
    PGN_TURBOCHARGER_WASTEGATE : UDINT := UDINT#16#FE96; (* < 65174 - TCW *)
    PGN_TURBOCHARGER_INFORMATION_5 : UDINT := UDINT#16#FE97; (* < 65175 - TCI5 *)
    PGN_TURBOCHARGER_INFORMATION_4 : UDINT := UDINT#16#FE98; (* < 65176 - TCI4 *)
    PGN_TURBOCHARGER_INFORMATION_3 : UDINT := UDINT#16#FE99; (* < 65177 - TCI3 *)
    PGN_TURBOCHARGER_INFORMATION_2 : UDINT := UDINT#16#FE9A; (* < 65178 - TCI2 *)
    PGN_TURBOCHARGER_INFORMATION_1 : UDINT := UDINT#16#FE9B; (* < 65179 - TCI1 *)
    PGN_MAIN_BEARING_TEMPERATURE_3 : UDINT := UDINT#16#FE9C; (* < 65180 - MBT3 *)
    PGN_MAIN_BEARING_TEMPERATURE_2 : UDINT := UDINT#16#FE9D; (* < 65181 - MBT2 *)
    PGN_MAIN_BEARING_TEMPERATURE_1 : UDINT := UDINT#16#FE9E; (* < 65182 - MBT1 *)
    PGN_EXHAUST_PORT_TEMPERATURE_5 : UDINT := UDINT#16#FE9F; (* < 65183 - EPT5 *)
    PGN_EXHAUST_PORT_TEMPERATURE_4 : UDINT := UDINT#16#FEA0; (* < 65184 - EPT4 *)
    PGN_EXHAUST_PORT_TEMPERATURE_3 : UDINT := UDINT#16#FEA1; (* < 65185 - EPT3 *)
    PGN_EXHAUST_PORT_TEMPERATURE_2 : UDINT := UDINT#16#FEA2; (* < 65186 - EPT2 *)
    PGN_EXHAUST_PORT_TEMPERATURE_1 : UDINT := UDINT#16#FEA3; (* < 65187 - EPT1 *)
    PGN_ENGINE_TEMPERATURE_2 : UDINT := UDINT#16#FEA4; (* < 65188 - ET2 *)
    PGN_INTAKE_MANIFOLD_INFO_2 : UDINT := UDINT#16#FEA5; (* < 65189 - IMT2 *)
    PGN_INTAKE_MANIFOLD_INFO_1 : UDINT := UDINT#16#FEA6; (* < 65190 - IMT1 *)
    PGN_ALTERNATE_FUEL_2 : UDINT := UDINT#16#FEA6; (* < 65190 - IMT1 *)
    PGN_ALTERNATOR_TEMPEATURE : UDINT := UDINT#16#FEA7; (* < 65191 - AT1 *)
    PGN_ARTICULATION_CONTROL : UDINT := UDINT#16#FEA8; (* < 65192 - ACTL *)
    PGN_EXHAUST_OXYGEN_1 : UDINT := UDINT#16#FEA9; (* < 65193 - EO1 *)
    PGN_ALTERNATE_FUEL_2_65194 : UDINT := UDINT#16#FEAA; (* < 65194 - AF2 *)
    PGN_ELECTRONIC_TRANSM_CONTR_6 : UDINT := UDINT#16#FEAB; (* < 65195 - ETC6 *)
    PGN_WHEEL_BRAKE_LIN_REMAIN_INFO : UDINT := UDINT#16#FEAC; (* < 65196 - EBC4 *)
    PGN_WHEEL_APPL_PRESS_HI_RGE_INF : UDINT := UDINT#16#FEAD; (* < 65197 - EBC3 *)
    PGN_AIR_SUPPLY_PRESSURE : UDINT := UDINT#16#FEAE; (* < 65198 - AIR1 *)
    PGN_FUEL_CONSUMPTION_GASEOUS : UDINT := UDINT#16#FEAF; (* < 65199 - GFC *)
    PGN_TRIP_TIME_INFORMATON_2 : UDINT := UDINT#16#FEB0; (* < 65200 - TTI2 *)
    PGN_ECU_HISTORY : UDINT := UDINT#16#FEB1; (* < 65201 - EH *)
    PGN_FUEL_INFORMATION_1_GASEOUS : UDINT := UDINT#16#FEB2; (* < 65202 - GFI1 *)
    PGN_FUEL_INFORMATION_LIQUID : UDINT := UDINT#16#FEB3; (* < 65203 - LFI1 *)
    PGN_TRIP_TIME_INFORMATION_1 : UDINT := UDINT#16#FEB4; (* < 65204 - TTI1 *)
    PGN_TRIP_SHUTDOWN_INFORMATION : UDINT := UDINT#16#FEB5; (* < 65205 - TSI *)
    PGN_TRIP_VEHIC_SPEED_DIST_INFO : UDINT := UDINT#16#FEB6; (* < 65206 - TVI *)
    PGN_ENGINE_SPEED_LOAD_FAC_INFO : UDINT := UDINT#16#FEB7; (* < 65207 - LF1 *)
    PGN_TRIP_FUEL_INFO_GASEOUS : UDINT := UDINT#16#FEB8; (* < 65208 - GTFI *)
    PGN_TRIP_FUEL_INFO_LIQUID : UDINT := UDINT#16#FEB9; (* < 65209 - LTFI *)
    PGN_TRIP_DISTANCE_INFO : UDINT := UDINT#16#FEBA; (* < 65210 - TDI *)
    PGN_TRIP_FAN_INFO : UDINT := UDINT#16#FEBB; (* < 65211 - TFI *)
    PGN_COMPRES_SERVICE_BRAKE_INFO : UDINT := UDINT#16#FEBC; (* < 65212 - CBI *)
    PGN_FAN_DRIVE : UDINT := UDINT#16#FEBD; (* < 65213 - FD1 *)
    PGN_ELECTRONIC_ENGIN_CONTROL_4 : UDINT := UDINT#16#FEBE; (* < 65214 - EEC4 *)
    PGN_WHEEL_SPEED_INFORMATION : UDINT := UDINT#16#FEBF; (* < 65215 - EBC2 *)
    PGN_SERVICE_INFORMATION : UDINT := UDINT#16#FEC0; (* < 65216 - SERV *)
    PGN_HIGH_RESOLUTION_VEHIC_DIST : UDINT := UDINT#16#FEC1; (* < 65217 - VDHR *)
    PGN_ELEC_RETARDER_CONTROLLER_2 : UDINT := UDINT#16#FEC2; (* < 65218 - ERC2 *)
    PGN_ELEC_TRANSMISSION_CONTR_5 : UDINT := UDINT#16#FEC3; (* < 65219 - ETC5 *)
    PGN_ELECTRONIC_BRAKE_SYSTEM_2_2 : UDINT := UDINT#16#FEC4; (* < 65220 - EBS22 *)
    PGN_ELEC_TRANSMISSION_CONTR_4 : UDINT := UDINT#16#FEC5; (* < 65221 - ETC4 *)
    PGN_ELECTRONIC_BRAKE_SYSTEM_2_3 : UDINT := UDINT#16#FEC6; (* < 65222 - EBS23 *)
    PGN_ELEC_TRANSMISSION_CONTR_3 : UDINT := UDINT#16#FEC7; (* < 65223 - ETC3 *)
    PGN_GENERAL_PURPOSE_MESSAGE_2_2 : UDINT := UDINT#16#FEC8; (* < 65224 - GPM22 *)
    PGN_ELECTRONIC_BRAKE_SYSTEM_1_2 : UDINT := UDINT#16#FEC9; (* < 65225 - EBS12 *)
    PGN_ACTIVE_DIAG_TROUBLE_CODES : UDINT := UDINT#16#FECA; (* < 65226 - DM1 *)
    PGN_PREV_ACTIV_DIAG_TROUBLE_COD : UDINT := UDINT#16#FECB; (* < 65227 - DM2 *)
    PGN_DIAGNOSTIC_DATA_CLEAR : UDINT := UDINT#16#FECC; (* < 65228 - DM3 *)
    PGN_FREEZE_FRAME_PARAMETERS : UDINT := UDINT#16#FECD; (* < 65229 - DM4 *)
    PGN_DIAGNOSTIC_READINESS : UDINT := UDINT#16#FECE; (* < 65230 - DM5 *)
    PGN_CONTIN_MONI_SYST_TEST_RESUL : UDINT := UDINT#16#FECF; (* < 65231 - DM6 *)
    PGN_TEST_RESUL_NON_CONT_MONITOR : UDINT := UDINT#16#FED0; (* < 65232 - DM8 *)
    PGN_OXYGEN_SENSOR_TEST_RESULTS : UDINT := UDINT#16#FED1; (* < 65233 - DM9 *)
    PGN_NON_CONTIN_MONITOR_SYS_TEST : UDINT := UDINT#16#FED2; (* < 65234 - DM10 *)
    PGN_DIAG_DATA_CLEAR_ACTIV_DTC : UDINT := UDINT#16#FED3; (* < 65235 - DM11 *)
    PGN_EMISS_RELAT_ACT_DIAG_TROUB : UDINT := UDINT#16#FED4; (* < 65236 - DM12 *)
    PGN_ALTERNATOR_SPEEED : UDINT := UDINT#16#FED5; (* < 65237 - AS1 *)
    PGN_HYBRID_OR_EV_SYSTEM_INPUTS_1 : UDINT := UDINT#16#FED6; (* < 65238 - HSI1 *)
    PGN_COMMANDED_ADDRESS : UDINT := UDINT#16#FED8; (* < 65240 - CA *)
    PGN_AUXIL_INPUT_OUTP_STATUS : UDINT := UDINT#16#FED9; (* < 65241 - AUXIO1 *)
    PGN_SOFTWARE_IDENTIFICATION : UDINT := UDINT#16#FEDA; (* < 65242 - SOFT *)
    PGN_ENGIN_FLUID_LEV_PRESSURE_2 : UDINT := UDINT#16#FEDB; (* < 65243 - EFL/P2 *)
    PGN_IDLE_OPERATION : UDINT := UDINT#16#FEDC; (* < 65244 - IO *)
    PGN_TURBOCHARGER : UDINT := UDINT#16#FEDD; (* < 65245 - TC *)
    PGN_AIR_START_PRESSURE : UDINT := UDINT#16#FEDE; (* < 65246 - AIR2 *)
    PGN_ELEC_ENGINE_CONTROLLER_3 : UDINT := UDINT#16#FEDF; (* < 65247 - EEC3 *)
    PGN_VEHICLE_DISTANCE : UDINT := UDINT#16#FEE0; (* < 65248 - VD *)
    PGN_RETARDER_CONFIGURATION : UDINT := UDINT#16#FEE1; (* < 65249 - RC *)
    PGN_TRANSMISSION_CONFIGURATION : UDINT := UDINT#16#FEE2; (* < 65250 - TCFG *)
    PGN_ENGINE_CONFIGURATION : UDINT := UDINT#16#FEE3; (* < 65251 - EC1 *)
    PGN_SHUTDOWN : UDINT := UDINT#16#FEE4; (* < 65252 - SHUTDN *)
    PGN_ENGINE_HOURS_REVOLUTIONS : UDINT := UDINT#16#FEE5; (* < 65253 - HOURS *)
    PGN_TIME_DATA : UDINT := UDINT#16#FEE6; (* < 65254 - TD *)
    PGN_VEHICLE_HOURS : UDINT := UDINT#16#FEE7; (* < 65255 - VH *)
    PGN_VEHICLE_DIRECTION_SPEED : UDINT := UDINT#16#FEE8; (* < 65256 - VDS *)
    PGN_FUEL_CONSUMPTION_LIQUID : UDINT := UDINT#16#FEE9; (* < 65257 - LFC1 *)
    PGN_VEHICLE_WEIGHT : UDINT := UDINT#16#FEEA; (* < 65258 - VW *)
    PGN_COMPONENT_IDENTIFICATION : UDINT := UDINT#16#FEEB; (* < 65259 - CI *)
    PGN_VEHICLE_IDENTIFICATION : UDINT := UDINT#16#FEEC; (* < 65260 - VI *)
    PGN_CRUIS_CTR_VEHIC_SPEED_SETUP : UDINT := UDINT#16#FEED; (* < 65261 - CCSS *)
    PGN_ENGINE_TEMPERATURE_1 : UDINT := UDINT#16#FEEE; (* < 65262 - ET1 *)
    PGN_ENGINE_FLUID_LEVEL_PRESS_1 : UDINT := UDINT#16#FEEF; (* < 65263 - EFL/P1 *)
    PGN_POWER_TAKEOFF_INFORMATION : UDINT := UDINT#16#FEF0; (* < 65264 - PTO1 *)
    PGN_CRUISE_CONTROL_VEHIC_SPEED : UDINT := UDINT#16#FEF1; (* < 65265 - CCVS1 *)
    PGN_FUEL_ECONOMY_LIQUID : UDINT := UDINT#16#FEF2; (* < 65266 - LFE1 *)
    PGN_VEHICLE_POSITION : UDINT := UDINT#16#FEF3; (* < 65267 - VP1 *)
    PGN_TIRE_CONDITION : UDINT := UDINT#16#FEF4; (* < 65268 - TIRE1 *)
    PGN_AMBIENT_CONDITIONS : UDINT := UDINT#16#FEF5; (* < 65269 - AMB *)
    PGN_INLET_EXHAUST_CONDITIONS_1 : UDINT := UDINT#16#FEF6; (* < 65270 - IC1 *)
    PGN_VEHICLE_ELECTRICAL_POWER : UDINT := UDINT#16#FEF7; (* < 65271 - VEP1 *)
    PGN_TRANSMISSION_FLUIDS : UDINT := UDINT#16#FEF8; (* < 65272 - TRF1 *)
    PGN_AXLE_INFORMATION : UDINT := UDINT#16#FEF9; (* < 65273 - AI *)
    PGN_BRAKES : UDINT := UDINT#16#FEFA; (* < 65274 - B1 *)
    PGN_RETARDER_FLUIDS : UDINT := UDINT#16#FEFB; (* < 65275 - RF *)
    PGN_DASH_DISPLAY : UDINT := UDINT#16#FEFC; (* < 65276 - DD1 *)
    PGN_ALTERNATE_FUEL_1 : UDINT := UDINT#16#FEFD; (* < 65277 - AF1 *)
    PGN_AUXIL_WATER_PUMP_PRESS : UDINT := UDINT#16#FEFE; (* < 65278 - AWPP *)
    PGN_WATER_IN_FUEL_INDICATOR : UDINT := UDINT#16#FEFF; (* < 65279 - OI *)
    PGN_PDU2_PropB : UDINT := UDINT#16#FF00; (* < 65280 - PropB_00 *)
    PGN_PROPRIETARY_B : UDINT := UDINT#16#FF01; (* < 65281 - PropB_01 *)
    PGN_PROPRIETARY_B_65282 : UDINT := UDINT#16#FF02; (* < 65282 - PropB_02 *)
    PGN_PROPRIETARY_B_65283 : UDINT := UDINT#16#FF03; (* < 65283 - PropB_03 *)
    PGN_PROPRIETARY_B_65284 : UDINT := UDINT#16#FF04; (* < 65284 - PropB_04 *)
    PGN_PROPRIETARY_B_65285 : UDINT := UDINT#16#FF05; (* < 65285 - PropB_05 *)
    PGN_PROPRIETARY_B_65286 : UDINT := UDINT#16#FF06; (* < 65286 - PropB_06 *)
    PGN_PROPRIETARY_B_65287 : UDINT := UDINT#16#FF07; (* < 65287 - PropB_07 *)
    PGN_PROPRIETARY_B_65288 : UDINT := UDINT#16#FF08; (* < 65288 - PropB_08 *)
    PGN_PROPRIETARY_B_65289 : UDINT := UDINT#16#FF09; (* < 65289 - PropB_09 *)
    PGN_PROPRIETARY_B_65290 : UDINT := UDINT#16#FF0A; (* < 65290 - PropB_0A *)
    PGN_PROPRIETARY_B_65291 : UDINT := UDINT#16#FF0B; (* < 65291 - PropB_0B *)
    PGN_PROPRIETARY_B_65292 : UDINT := UDINT#16#FF0C; (* < 65292 - PropB_0C *)
    PGN_PROPRIETARY_B_65293 : UDINT := UDINT#16#FF0D; (* < 65293 - PropB_0D *)
    PGN_PROPRIETARY_B_65294 : UDINT := UDINT#16#FF0E; (* < 65294 - PropB_0E *)
    PGN_PROPRIETARY_B_65295 : UDINT := UDINT#16#FF0F; (* < 65295 - PropB_0F *)
    PGN_PROPRIETARY_B_65296 : UDINT := UDINT#16#FF10; (* < 65296 - PropB_10 *)
    PGN_PROPRIETARY_B_65297 : UDINT := UDINT#16#FF11; (* < 65297 - PropB_11 *)
    PGN_PROPRIETARY_B_65298 : UDINT := UDINT#16#FF12; (* < 65298 - PropB_12 *)
    PGN_PROPRIETARY_B_65299 : UDINT := UDINT#16#FF13; (* < 65299 - PropB_13 *)
    PGN_PROPRIETARY_B_65300 : UDINT := UDINT#16#FF14; (* < 65300 - PropB_14 *)
    PGN_PROPRIETARY_B_65301 : UDINT := UDINT#16#FF15; (* < 65301 - PropB_15 *)
    PGN_PROPRIETARY_B_65302 : UDINT := UDINT#16#FF16; (* < 65302 - PropB_16 *)
    PGN_PROPRIETARY_B_65303 : UDINT := UDINT#16#FF17; (* < 65303 - PropB_17 *)
    PGN_PROPRIETARY_B_65304 : UDINT := UDINT#16#FF18; (* < 65304 - PropB_18 *)
    PGN_PROPRIETARY_B_65305 : UDINT := UDINT#16#FF19; (* < 65305 - PropB_19 *)
    PGN_PROPRIETARY_B_65306 : UDINT := UDINT#16#FF1A; (* < 65306 - PropB_1A *)
    PGN_PROPRIETARY_B_65307 : UDINT := UDINT#16#FF1B; (* < 65307 - PropB_1B *)
    PGN_PROPRIETARY_B_65308 : UDINT := UDINT#16#FF1C; (* < 65308 - PropB_1C *)
    PGN_PROPRIETARY_B_65309 : UDINT := UDINT#16#FF1D; (* < 65309 - PropB_1D *)
    PGN_PROPRIETARY_B_65310 : UDINT := UDINT#16#FF1E; (* < 65310 - PropB_1E *)
    PGN_PROPRIETARY_B_65311 : UDINT := UDINT#16#FF1F; (* < 65311 - PropB_1F *)
    PGN_PROPRIETARY_B_65312 : UDINT := UDINT#16#FF20; (* < 65312 - PropB_20 *)
    PGN_PROPRIETARY_B_65313 : UDINT := UDINT#16#FF21; (* < 65313 - PropB_21 *)
    PGN_PROPRIETARY_B_65314 : UDINT := UDINT#16#FF22; (* < 65314 - PropB_22 *)
    PGN_PROPRIETARY_B_65315 : UDINT := UDINT#16#FF23; (* < 65315 - PropB_23 *)
    PGN_PROPRIETARY_B_65316 : UDINT := UDINT#16#FF24; (* < 65316 - PropB_24 *)
    PGN_PROPRIETARY_B_65317 : UDINT := UDINT#16#FF25; (* < 65317 - PropB_25 *)
    PGN_PROPRIETARY_B_65318 : UDINT := UDINT#16#FF26; (* < 65318 - PropB_26 *)
    PGN_PROPRIETARY_B_65319 : UDINT := UDINT#16#FF27; (* < 65319 - PropB_27 *)
    PGN_PROPRIETARY_B_65320 : UDINT := UDINT#16#FF28; (* < 65320 - PropB_28 *)
    PGN_PROPRIETARY_B_65321 : UDINT := UDINT#16#FF29; (* < 65321 - PropB_29 *)
    PGN_PROPRIETARY_B_65322 : UDINT := UDINT#16#FF2A; (* < 65322 - PropB_2A *)
    PGN_PROPRIETARY_B_65323 : UDINT := UDINT#16#FF2B; (* < 65323 - PropB_2B *)
    PGN_PROPRIETARY_B_65324 : UDINT := UDINT#16#FF2C; (* < 65324 - PropB_2C *)
    PGN_PROPRIETARY_B_65325 : UDINT := UDINT#16#FF2D; (* < 65325 - PropB_2D *)
    PGN_PROPRIETARY_B_65326 : UDINT := UDINT#16#FF2E; (* < 65326 - PropB_2E *)
    PGN_PROPRIETARY_B_65327 : UDINT := UDINT#16#FF2F; (* < 65327 - PropB_2F *)
    PGN_PROPRIETARY_B_65328 : UDINT := UDINT#16#FF30; (* < 65328 - PropB_30 *)
    PGN_PROPRIETARY_B_65329 : UDINT := UDINT#16#FF31; (* < 65329 - PropB_31 *)
    PGN_PROPRIETARY_B_65330 : UDINT := UDINT#16#FF32; (* < 65330 - PropB_32 *)
    PGN_PROPRIETARY_B_65331 : UDINT := UDINT#16#FF33; (* < 65331 - PropB_33 *)
    PGN_PROPRIETARY_B_65332 : UDINT := UDINT#16#FF34; (* < 65332 - PropB_34 *)
    PGN_PROPRIETARY_B_65333 : UDINT := UDINT#16#FF35; (* < 65333 - PropB_35 *)
    PGN_PROPRIETARY_B_65334 : UDINT := UDINT#16#FF36; (* < 65334 - PropB_36 *)
    PGN_PROPRIETARY_B_65335 : UDINT := UDINT#16#FF37; (* < 65335 - PropB_37 *)
    PGN_PROPRIETARY_B_65336 : UDINT := UDINT#16#FF38; (* < 65336 - PropB_38 *)
    PGN_PROPRIETARY_B_65337 : UDINT := UDINT#16#FF39; (* < 65337 - PropB_39 *)
    PGN_PROPRIETARY_B_65338 : UDINT := UDINT#16#FF3A; (* < 65338 - PropB_3A *)
    PGN_PROPRIETARY_B_65339 : UDINT := UDINT#16#FF3B; (* < 65339 - PropB_3B *)
    PGN_PROPRIETARY_B_65340 : UDINT := UDINT#16#FF3C; (* < 65340 - PropB_3C *)
    PGN_PROPRIETARY_B_65341 : UDINT := UDINT#16#FF3D; (* < 65341 - PropB_3D *)
    PGN_PROPRIETARY_B_65342 : UDINT := UDINT#16#FF3E; (* < 65342 - PropB_3E *)
    PGN_PROPRIETARY_B_65343 : UDINT := UDINT#16#FF3F; (* < 65343 - PropB_3F *)
    PGN_PROPRIETARY_B_65344 : UDINT := UDINT#16#FF40; (* < 65344 - PropB_40 *)
    PGN_PROPRIETARY_B_65345 : UDINT := UDINT#16#FF41; (* < 65345 - PropB_41 *)
    PGN_PROPRIETARY_B_65346 : UDINT := UDINT#16#FF42; (* < 65346 - PropB_42 *)
    PGN_PROPRIETARY_B_65347 : UDINT := UDINT#16#FF43; (* < 65347 - PropB_43 *)
    PGN_PROPRIETARY_B_65348 : UDINT := UDINT#16#FF44; (* < 65348 - PropB_44 *)
    PGN_PROPRIETARY_B_65349 : UDINT := UDINT#16#FF45; (* < 65349 - PropB_45 *)
    PGN_PROPRIETARY_B_65350 : UDINT := UDINT#16#FF46; (* < 65350 - PropB_46 *)
    PGN_PROPRIETARY_B_65351 : UDINT := UDINT#16#FF47; (* < 65351 - PropB_47 *)
    PGN_PROPRIETARY_B_65352 : UDINT := UDINT#16#FF48; (* < 65352 - PropB_48 *)
    PGN_PROPRIETARY_B_65353 : UDINT := UDINT#16#FF49; (* < 65353 - PropB_49 *)
    PGN_PROPRIETARY_B_65354 : UDINT := UDINT#16#FF4A; (* < 65354 - PropB_4A *)
    PGN_PROPRIETARY_B_65355 : UDINT := UDINT#16#FF4B; (* < 65355 - PropB_4B *)
    PGN_PROPRIETARY_B_65356 : UDINT := UDINT#16#FF4C; (* < 65356 - PropB_4C *)
    PGN_PROPRIETARY_B_65357 : UDINT := UDINT#16#FF4D; (* < 65357 - PropB_4D *)
    PGN_PROPRIETARY_B_65358 : UDINT := UDINT#16#FF4E; (* < 65358 - PropB_4E *)
    PGN_PROPRIETARY_B_65359 : UDINT := UDINT#16#FF4F; (* < 65359 - PropB_4F *)
    PGN_PROPRIETARY_B_65360 : UDINT := UDINT#16#FF50; (* < 65360 - PropB_50 *)
    PGN_PROPRIETARY_B_65361 : UDINT := UDINT#16#FF51; (* < 65361 - PropB_51 *)
    PGN_PROPRIETARY_B_65362 : UDINT := UDINT#16#FF52; (* < 65362 - PropB_52 *)
    PGN_PROPRIETARY_B_65363 : UDINT := UDINT#16#FF53; (* < 65363 - PropB_53 *)
    PGN_PROPRIETARY_B_65364 : UDINT := UDINT#16#FF54; (* < 65364 - PropB_54 *)
    PGN_PROPRIETARY_B_65365 : UDINT := UDINT#16#FF55; (* < 65365 - PropB_55 *)
    PGN_PROPRIETARY_B_65366 : UDINT := UDINT#16#FF56; (* < 65366 - PropB_56 *)
    PGN_PROPRIETARY_B_65367 : UDINT := UDINT#16#FF57; (* < 65367 - PropB_57 *)
    PGN_PROPRIETARY_B_65368 : UDINT := UDINT#16#FF58; (* < 65368 - PropB_58 *)
    PGN_PROPRIETARY_B_65369 : UDINT := UDINT#16#FF59; (* < 65369 - PropB_59 *)
    PGN_PROPRIETARY_B_65370 : UDINT := UDINT#16#FF5A; (* < 65370 - PropB_5A *)
    PGN_PROPRIETARY_B_65371 : UDINT := UDINT#16#FF5B; (* < 65371 - PropB_5B *)
    PGN_PROPRIETARY_B_65372 : UDINT := UDINT#16#FF5C; (* < 65372 - PropB_5C *)
    PGN_PROPRIETARY_B_65373 : UDINT := UDINT#16#FF5D; (* < 65373 - PropB_5D *)
    PGN_PROPRIETARY_B_65374 : UDINT := UDINT#16#FF5E; (* < 65374 - PropB_5E *)
    PGN_PROPRIETARY_B_65375 : UDINT := UDINT#16#FF5F; (* < 65375 - PropB_5F *)
    PGN_PROPRIETARY_B_65376 : UDINT := UDINT#16#FF60; (* < 65376 - PropB_60 *)
    PGN_PROPRIETARY_B_65377 : UDINT := UDINT#16#FF61; (* < 65377 - PropB_61 *)
    PGN_PROPRIETARY_B_65378 : UDINT := UDINT#16#FF62; (* < 65378 - PropB_62 *)
    PGN_PROPRIETARY_B_65379 : UDINT := UDINT#16#FF63; (* < 65379 - PropB_63 *)
    PGN_PROPRIETARY_B_65380 : UDINT := UDINT#16#FF64; (* < 65380 - PropB_64 *)
    PGN_PROPRIETARY_B_65381 : UDINT := UDINT#16#FF65; (* < 65381 - PropB_65 *)
    PGN_PROPRIETARY_B_65382 : UDINT := UDINT#16#FF66; (* < 65382 - PropB_66 *)
    PGN_PROPRIETARY_B_65383 : UDINT := UDINT#16#FF67; (* < 65383 - PropB_67 *)
    PGN_PROPRIETARY_B_65384 : UDINT := UDINT#16#FF68; (* < 65384 - PropB_68 *)
    PGN_PROPRIETARY_B_65385 : UDINT := UDINT#16#FF69; (* < 65385 - PropB_69 *)
    PGN_PROPRIETARY_B_65386 : UDINT := UDINT#16#FF6A; (* < 65386 - PropB_6A *)
    PGN_PROPRIETARY_B_65387 : UDINT := UDINT#16#FF6B; (* < 65387 - PropB_6B *)
    PGN_PROPRIETARY_B_65388 : UDINT := UDINT#16#FF6C; (* < 65388 - PropB_6C *)
    PGN_PROPRIETARY_B_65389 : UDINT := UDINT#16#FF6D; (* < 65389 - PropB_6D *)
    PGN_PROPRIETARY_B_65390 : UDINT := UDINT#16#FF6E; (* < 65390 - PropB_6E *)
    PGN_PROPRIETARY_B_65391 : UDINT := UDINT#16#FF6F; (* < 65391 - PropB_6F *)
    PGN_PROPRIETARY_B_65392 : UDINT := UDINT#16#FF70; (* < 65392 - PropB_70 *)
    PGN_PROPRIETARY_B_65393 : UDINT := UDINT#16#FF71; (* < 65393 - PropB_71 *)
    PGN_PROPRIETARY_B_65394 : UDINT := UDINT#16#FF72; (* < 65394 - PropB_72 *)
    PGN_PROPRIETARY_B_65395 : UDINT := UDINT#16#FF73; (* < 65395 - PropB_73 *)
    PGN_PROPRIETARY_B_65396 : UDINT := UDINT#16#FF74; (* < 65396 - PropB_74 *)
    PGN_PROPRIETARY_B_65397 : UDINT := UDINT#16#FF75; (* < 65397 - PropB_75 *)
    PGN_PROPRIETARY_B_65398 : UDINT := UDINT#16#FF76; (* < 65398 - PropB_76 *)
    PGN_PROPRIETARY_B_65399 : UDINT := UDINT#16#FF77; (* < 65399 - PropB_77 *)
    PGN_PROPRIETARY_B_65400 : UDINT := UDINT#16#FF78; (* < 65400 - PropB_78 *)
    PGN_PROPRIETARY_B_65401 : UDINT := UDINT#16#FF79; (* < 65401 - PropB_79 *)
    PGN_PROPRIETARY_B_65402 : UDINT := UDINT#16#FF7A; (* < 65402 - PropB_7A *)
    PGN_PROPRIETARY_B_65403 : UDINT := UDINT#16#FF7B; (* < 65403 - PropB_7B *)
    PGN_PROPRIETARY_B_65404 : UDINT := UDINT#16#FF7C; (* < 65404 - PropB_7C *)
    PGN_PROPRIETARY_B_65405 : UDINT := UDINT#16#FF7D; (* < 65405 - PropB_7D *)
    PGN_PROPRIETARY_B_65406 : UDINT := UDINT#16#FF7E; (* < 65406 - PropB_7E *)
    PGN_PROPRIETARY_B_65407 : UDINT := UDINT#16#FF7F; (* < 65407 - PropB_7F *)
    PGN_PROPRIETARY_B_65408 : UDINT := UDINT#16#FF80; (* < 65408 - PropB_80 *)
    PGN_PROPRIETARY_B_65409 : UDINT := UDINT#16#FF81; (* < 65409 - PropB_81 *)
    PGN_PROPRIETARY_B_65410 : UDINT := UDINT#16#FF82; (* < 65410 - PropB_82 *)
    PGN_PROPRIETARY_B_65411 : UDINT := UDINT#16#FF83; (* < 65411 - PropB_83 *)
    PGN_PROPRIETARY_B_65412 : UDINT := UDINT#16#FF84; (* < 65412 - PropB_84 *)
    PGN_PROPRIETARY_B_65413 : UDINT := UDINT#16#FF85; (* < 65413 - PropB_85 *)
    PGN_PROPRIETARY_B_65414 : UDINT := UDINT#16#FF86; (* < 65414 - PropB_86 *)
    PGN_PROPRIETARY_B_65415 : UDINT := UDINT#16#FF87; (* < 65415 - PropB_87 *)
    PGN_PROPRIETARY_B_65416 : UDINT := UDINT#16#FF88; (* < 65416 - PropB_88 *)
    PGN_PROPRIETARY_B_65417 : UDINT := UDINT#16#FF89; (* < 65417 - PropB_89 *)
    PGN_PROPRIETARY_B_65418 : UDINT := UDINT#16#FF8A; (* < 65418 - PropB_8A *)
    PGN_PROPRIETARY_B_65419 : UDINT := UDINT#16#FF8B; (* < 65419 - PropB_8B *)
    PGN_PROPRIETARY_B_65420 : UDINT := UDINT#16#FF8C; (* < 65420 - PropB_8C *)
    PGN_PROPRIETARY_B_65421 : UDINT := UDINT#16#FF8D; (* < 65421 - PropB_8D *)
    PGN_PROPRIETARY_B_65422 : UDINT := UDINT#16#FF8E; (* < 65422 - PropB_8E *)
    PGN_PROPRIETARY_B_65423 : UDINT := UDINT#16#FF8F; (* < 65423 - PropB_8F *)
    PGN_PROPRIETARY_B_65424 : UDINT := UDINT#16#FF90; (* < 65424 - PropB_90 *)
    PGN_PROPRIETARY_B_65425 : UDINT := UDINT#16#FF91; (* < 65425 - PropB_91 *)
    PGN_PROPRIETARY_B_65426 : UDINT := UDINT#16#FF92; (* < 65426 - PropB_92 *)
    PGN_PROPRIETARY_B_65427 : UDINT := UDINT#16#FF93; (* < 65427 - PropB_93 *)
    PGN_PROPRIETARY_B_65428 : UDINT := UDINT#16#FF94; (* < 65428 - PropB_94 *)
    PGN_PROPRIETARY_B_65429 : UDINT := UDINT#16#FF95; (* < 65429 - PropB_95 *)
    PGN_PROPRIETARY_B_65430 : UDINT := UDINT#16#FF96; (* < 65430 - PropB_96 *)
    PGN_PROPRIETARY_B_65431 : UDINT := UDINT#16#FF97; (* < 65431 - PropB_97 *)
    PGN_PROPRIETARY_B_65432 : UDINT := UDINT#16#FF98; (* < 65432 - PropB_98 *)
    PGN_PROPRIETARY_B_65433 : UDINT := UDINT#16#FF99; (* < 65433 - PropB_99 *)
    PGN_PROPRIETARY_B_65434 : UDINT := UDINT#16#FF9A; (* < 65434 - PropB_9A *)
    PGN_PROPRIETARY_B_65435 : UDINT := UDINT#16#FF9B; (* < 65435 - PropB_9B *)
    PGN_PROPRIETARY_B_65436 : UDINT := UDINT#16#FF9C; (* < 65436 - PropB_9C *)
    PGN_PROPRIETARY_B_65437 : UDINT := UDINT#16#FF9D; (* < 65437 - PropB_9D *)
    PGN_PROPRIETARY_B_65438 : UDINT := UDINT#16#FF9E; (* < 65438 - PropB_9E *)
    PGN_PROPRIETARY_B_65439 : UDINT := UDINT#16#FF9F; (* < 65439 - PropB_9F *)
    PGN_PROPRIETARY_B_65440 : UDINT := UDINT#16#FFA0; (* < 65440 - PropB_A0 *)
    PGN_PROPRIETARY_B_65441 : UDINT := UDINT#16#FFA1; (* < 65441 - PropB_A1 *)
    PGN_PROPRIETARY_B_65442 : UDINT := UDINT#16#FFA2; (* < 65442 - PropB_A2 *)
    PGN_PROPRIETARY_B_65443 : UDINT := UDINT#16#FFA3; (* < 65443 - PropB_A3 *)
    PGN_PROPRIETARY_B_65444 : UDINT := UDINT#16#FFA4; (* < 65444 - PropB_A4 *)
    PGN_PROPRIETARY_B_65445 : UDINT := UDINT#16#FFA5; (* < 65445 - PropB_A5 *)
    PGN_PROPRIETARY_B_65446 : UDINT := UDINT#16#FFA6; (* < 65446 - PropB_A6 *)
    PGN_PROPRIETARY_B_65447 : UDINT := UDINT#16#FFA7; (* < 65447 - PropB_A7 *)
    PGN_PROPRIETARY_B_65448 : UDINT := UDINT#16#FFA8; (* < 65448 - PropB_A8 *)
    PGN_PROPRIETARY_B_65449 : UDINT := UDINT#16#FFA9; (* < 65449 - PropB_A9 *)
    PGN_PROPRIETARY_B_65450 : UDINT := UDINT#16#FFAA; (* < 65450 - PropB_AA *)
    PGN_PROPRIETARY_B_65451 : UDINT := UDINT#16#FFAB; (* < 65451 - PropB_AB *)
    PGN_PROPRIETARY_B_65452 : UDINT := UDINT#16#FFAC; (* < 65452 - PropB_AC *)
    PGN_PROPRIETARY_B_65453 : UDINT := UDINT#16#FFAD; (* < 65453 - PropB_AD *)
    PGN_PROPRIETARY_B_65454 : UDINT := UDINT#16#FFAE; (* < 65454 - PropB_AE *)
    PGN_PROPRIETARY_B_65455 : UDINT := UDINT#16#FFAF; (* < 65455 - PropB_AF *)
    PGN_PROPRIETARY_B_65456 : UDINT := UDINT#16#FFB0; (* < 65456 - PropB_B0 *)
    PGN_PROPRIETARY_B_65457 : UDINT := UDINT#16#FFB1; (* < 65457 - PropB_B1 *)
    PGN_PROPRIETARY_B_65458 : UDINT := UDINT#16#FFB2; (* < 65458 - PropB_B2 *)
    PGN_PROPRIETARY_B_65459 : UDINT := UDINT#16#FFB3; (* < 65459 - PropB_B3 *)
    PGN_PROPRIETARY_B_65460 : UDINT := UDINT#16#FFB4; (* < 65460 - PropB_B4 *)
    PGN_PROPRIETARY_B_65461 : UDINT := UDINT#16#FFB5; (* < 65461 - PropB_B5 *)
    PGN_PROPRIETARY_B_65462 : UDINT := UDINT#16#FFB6; (* < 65462 - PropB_B6 *)
    PGN_PROPRIETARY_B_65463 : UDINT := UDINT#16#FFB7; (* < 65463 - PropB_B7 *)
    PGN_PROPRIETARY_B_65464 : UDINT := UDINT#16#FFB8; (* < 65464 - PropB_B8 *)
    PGN_PROPRIETARY_B_65465 : UDINT := UDINT#16#FFB9; (* < 65465 - PropB_B9 *)
    PGN_PROPRIETARY_B_65466 : UDINT := UDINT#16#FFBA; (* < 65466 - PropB_BA *)
    PGN_PROPRIETARY_B_65467 : UDINT := UDINT#16#FFBB; (* < 65467 - PropB_BB *)
    PGN_PROPRIETARY_B_65468 : UDINT := UDINT#16#FFBC; (* < 65468 - PropB_BC *)
    PGN_PROPRIETARY_B_65469 : UDINT := UDINT#16#FFBD; (* < 65469 - PropB_BD *)
    PGN_PROPRIETARY_B_65470 : UDINT := UDINT#16#FFBE; (* < 65470 - PropB_BE *)
    PGN_PROPRIETARY_B_65471 : UDINT := UDINT#16#FFBF; (* < 65471 - PropB_BF *)
    PGN_PROPRIETARY_B_65472 : UDINT := UDINT#16#FFC0; (* < 65472 - PropB_C0 *)
    PGN_PROPRIETARY_B_65473 : UDINT := UDINT#16#FFC1; (* < 65473 - PropB_C1 *)
    PGN_PROPRIETARY_B_65474 : UDINT := UDINT#16#FFC2; (* < 65474 - PropB_C2 *)
    PGN_PROPRIETARY_B_65475 : UDINT := UDINT#16#FFC3; (* < 65475 - PropB_C3 *)
    PGN_PROPRIETARY_B_65476 : UDINT := UDINT#16#FFC4; (* < 65476 - PropB_C4 *)
    PGN_PROPRIETARY_B_65477 : UDINT := UDINT#16#FFC5; (* < 65477 - PropB_C5 *)
    PGN_PROPRIETARY_B_65478 : UDINT := UDINT#16#FFC6; (* < 65478 - PropB_C6 *)
    PGN_PROPRIETARY_B_65479 : UDINT := UDINT#16#FFC7; (* < 65479 - PropB_C7 *)
    PGN_PROPRIETARY_B_65480 : UDINT := UDINT#16#FFC8; (* < 65480 - PropB_C8 *)
    PGN_PROPRIETARY_B_65481 : UDINT := UDINT#16#FFC9; (* < 65481 - PropB_C9 *)
    PGN_PROPRIETARY_B_65482 : UDINT := UDINT#16#FFCA; (* < 65482 - PropB_CA *)
    PGN_PROPRIETARY_B_65483 : UDINT := UDINT#16#FFCB; (* < 65483 - PropB_CB *)
    PGN_PROPRIETARY_B_65484 : UDINT := UDINT#16#FFCC; (* < 65484 - PropB_CC *)
    PGN_PROPRIETARY_B_65485 : UDINT := UDINT#16#FFCD; (* < 65485 - PropB_CD *)
    PGN_PROPRIETARY_B_65486 : UDINT := UDINT#16#FFCE; (* < 65486 - PropB_CE *)
    PGN_PROPRIETARY_B_65487 : UDINT := UDINT#16#FFCF; (* < 65487 - PropB_CF *)
    PGN_PROPRIETARY_B_65488 : UDINT := UDINT#16#FFD0; (* < 65488 - PropB_D0 *)
    PGN_PROPRIETARY_B_65489 : UDINT := UDINT#16#FFD1; (* < 65489 - PropB_D1 *)
    PGN_PROPRIETARY_B_65490 : UDINT := UDINT#16#FFD2; (* < 65490 - PropB_D2 *)
    PGN_PROPRIETARY_B_65491 : UDINT := UDINT#16#FFD3; (* < 65491 - PropB_D3 *)
    PGN_PROPRIETARY_B_65492 : UDINT := UDINT#16#FFD4; (* < 65492 - PropB_D4 *)
    PGN_PROPRIETARY_B_65493 : UDINT := UDINT#16#FFD5; (* < 65493 - PropB_D5 *)
    PGN_PROPRIETARY_B_65494 : UDINT := UDINT#16#FFD6; (* < 65494 - PropB_D6 *)
    PGN_PROPRIETARY_B_65495 : UDINT := UDINT#16#FFD7; (* < 65495 - PropB_D7 *)
    PGN_PROPRIETARY_B_65496 : UDINT := UDINT#16#FFD8; (* < 65496 - PropB_D8 *)
    PGN_PROPRIETARY_B_65497 : UDINT := UDINT#16#FFD9; (* < 65497 - PropB_D9 *)
    PGN_PROPRIETARY_B_65498 : UDINT := UDINT#16#FFDA; (* < 65498 - PropB_DA *)
    PGN_PROPRIETARY_B_65499 : UDINT := UDINT#16#FFDB; (* < 65499 - PropB_DB *)
    PGN_PROPRIETARY_B_65500 : UDINT := UDINT#16#FFDC; (* < 65500 - PropB_DC *)
    PGN_PROPRIETARY_B_65501 : UDINT := UDINT#16#FFDD; (* < 65501 - PropB_DD *)
    PGN_PROPRIETARY_B_65502 : UDINT := UDINT#16#FFDE; (* < 65502 - PropB_DE *)
    PGN_PROPRIETARY_B_65503 : UDINT := UDINT#16#FFDF; (* < 65503 - PropB_DF *)
    PGN_PROPRIETARY_B_65504 : UDINT := UDINT#16#FFE0; (* < 65504 - PropB_E0 *)
    PGN_PROPRIETARY_B_65505 : UDINT := UDINT#16#FFE1; (* < 65505 - PropB_E1 *)
    PGN_PROPRIETARY_B_65506 : UDINT := UDINT#16#FFE2; (* < 65506 - PropB_E2 *)
    PGN_PROPRIETARY_B_65507 : UDINT := UDINT#16#FFE3; (* < 65507 - PropB_E3 *)
    PGN_PROPRIETARY_B_65508 : UDINT := UDINT#16#FFE4; (* < 65508 - PropB_E4 *)
    PGN_PROPRIETARY_B_65509 : UDINT := UDINT#16#FFE5; (* < 65509 - PropB_E5 *)
    PGN_PROPRIETARY_B_65510 : UDINT := UDINT#16#FFE6; (* < 65510 - PropB_E6 *)
    PGN_PROPRIETARY_B_65511 : UDINT := UDINT#16#FFE7; (* < 65511 - PropB_E7 *)
    PGN_PROPRIETARY_B_65512 : UDINT := UDINT#16#FFE8; (* < 65512 - PropB_E8 *)
    PGN_PROPRIETARY_B_65513 : UDINT := UDINT#16#FFE9; (* < 65513 - PropB_E9 *)
    PGN_PROPRIETARY_B_65514 : UDINT := UDINT#16#FFEA; (* < 65514 - PropB_EA *)
    PGN_PROPRIETARY_B_65515 : UDINT := UDINT#16#FFEB; (* < 65515 - PropB_EB *)
    PGN_PROPRIETARY_B_65516 : UDINT := UDINT#16#FFEC; (* < 65516 - PropB_EC *)
    PGN_PROPRIETARY_B_65517 : UDINT := UDINT#16#FFED; (* < 65517 - PropB_ED *)
    PGN_PROPRIETARY_B_65518 : UDINT := UDINT#16#FFEE; (* < 65518 - PropB_EE *)
    PGN_PROPRIETARY_B_65519 : UDINT := UDINT#16#FFEF; (* < 65519 - PropB_EF *)
    PGN_PROPRIETARY_B_65520 : UDINT := UDINT#16#FFF0; (* < 65520 - PropB_F0 *)
    PGN_PROPRIETARY_B_65521 : UDINT := UDINT#16#FFF1; (* < 65521 - PropB_F1 *)
    PGN_PROPRIETARY_B_65522 : UDINT := UDINT#16#FFF2; (* < 65522 - PropB_F2 *)
    PGN_PROPRIETARY_B_65523 : UDINT := UDINT#16#FFF3; (* < 65523 - PropB_F3 *)
    PGN_PROPRIETARY_B_65524 : UDINT := UDINT#16#FFF4; (* < 65524 - PropB_F4 *)
    PGN_PROPRIETARY_B_65525 : UDINT := UDINT#16#FFF5; (* < 65525 - PropB_F5 *)
    PGN_PROPRIETARY_B_65526 : UDINT := UDINT#16#FFF6; (* < 65526 - PropB_F6 *)
    PGN_PROPRIETARY_B_65527 : UDINT := UDINT#16#FFF7; (* < 65527 - PropB_F7 *)
    PGN_PROPRIETARY_B_65528 : UDINT := UDINT#16#FFF8; (* < 65528 - PropB_F8 *)
    PGN_PROPRIETARY_B_65529 : UDINT := UDINT#16#FFF9; (* < 65529 - PropB_F9 *)
    PGN_PROPRIETARY_B_65530 : UDINT := UDINT#16#FFFA; (* < 65530 - PropB_FA *)
    PGN_PROPRIETARY_B_65531 : UDINT := UDINT#16#FFFB; (* < 65531 - PropB_FB *)
    PGN_PROPRIETARY_B_65532 : UDINT := UDINT#16#FFFC; (* < 65532 - PropB_FC *)
    PGN_PROPRIETARY_B_65533 : UDINT := UDINT#16#FFFD; (* < 65533 - PropB_FD *)
    PGN_PROPRIETARY_B_65534 : UDINT := UDINT#16#FFFE; (* < 65534 - PropB_FE *)
    PGN_PROPRIETARY_B_LAST_ENTRY : UDINT := UDINT#16#FFFF; (* < 65535 - PropB_FF *)
    PGN_NMEA_REQCMDACKGROUPFUNCION : UDINT := UDINT#16#1ED00; (* < 126208 - NMEA - Request/Command/Acknowledge group function *)
    PGN_PGNLIST_GROUPFUNCTION : UDINT := UDINT#16#1EE00; (* < 126464 - PGN List - Transmit/Receive PGN's group function *)
    PGN_PDU1_PropA2 : UDINT := UDINT#16#1EF00; (* < 126720 - PropA2 *)
    PGN_ALERT : UDINT := UDINT#16#1F007; (* < 126983 - Alert *)
    PGN_ALERT_RESPONSE : UDINT := UDINT#16#1F008; (* < 126984 - Alert Response *)
    PGN_ALERT_TEXT : UDINT := UDINT#16#1F009; (* < 126985 - Alert Text *)
    PGN_ALERT_CONFIGURATION : UDINT := UDINT#16#1F00A; (* < 126986 - Alert Configuration *)
    PGN_ALERT_THRESHOLD : UDINT := UDINT#16#1F00B; (* < 126987 - Alert Threshold *)
    PGN_ALERT_VALUE : UDINT := UDINT#16#1F00C; (* < 126988 - Alert Value *)
    PGN_SYTEMTIME : UDINT := UDINT#16#1F010; (* < 126992 - System Time *)
    PGN_HEARTBEAT_126993 : UDINT := UDINT#16#1F011; (* < 126993 - Heartbeat *)
    PGN_PRODUKTINFORMATION : UDINT := UDINT#16#1F014; (* < 126996 - Product Information *)
    PGN_CONFIGURATIONINFORMATION : UDINT := UDINT#16#1F016; (* < 126998 - Configuration Information *)
    PGN_CYCLIC_ALERT_LIST_IEC_61924_2 : UDINT := UDINT#16#1F019; (* < 127001 - Cyclic Alert List - IEC 61924-2 *)
    PGN_RESPONSIBILITY_TRANSFER_FUNCTION_IEC_61924_2 : UDINT := UDINT#16#1F01A; (* < 127002 - Responsibility Transfer Function - IEC 61924-2 *)
    PGN_MAN_OVERBOARD_NOTIFICATION_MOB : UDINT := UDINT#16#1F101; (* < 127233 - Man Overboard Notification (MOB) *)
    PGN_HEADING_TRACKCONTROL : UDINT := UDINT#16#1F105; (* < 127237 - Heading/Track Control *)
    PGN_RUDDER : UDINT := UDINT#16#1F10D; (* < 127245 - Rudder *)
    PGN_VESSEL_HEADING : UDINT := UDINT#16#1F112; (* < 127250 - Vessel Heading *)
    PGN_RATE_OF_TURN : UDINT := UDINT#16#1F113; (* < 127251 - Rate of Turn *)
    PGN_HEAVE : UDINT := UDINT#16#1F114; (* < 127252 - Heave *)
    PGN_ATTITUDE : UDINT := UDINT#16#1F119; (* < 127257 - Attitude *)
    PGN_MAGNETIC_VARIATION : UDINT := UDINT#16#1F11A; (* < 127258 - Magnetic Variation *)
    PGN_ENGINE_PARA_RAPID_UPDATE : UDINT := UDINT#16#1F200; (* < 127488 - Engine Parameters, Rapid Update *)
    PGN_ENGINE_PARA_DYNAMIC : UDINT := UDINT#16#1F201; (* < 127489 - Engine Parameters, Dynamic *)
    PGN_ELECTRIC_DRIVE_STATUS_DYNAMIC : UDINT := UDINT#16#1F202; (* < 127490 - Electric Drive Status, Dynamic *)
    PGN_ELECTRIC_ENERGY_STORAGE_STATUS_DYNAMIC : UDINT := UDINT#16#1F203; (* < 127491 - Electric Energy Storage Status, Dynamic *)
    PGN_TRANSMISSION_PARA_DYNAMIC : UDINT := UDINT#16#1F205; (* < 127493 - Transmission Parameters, Dynamic *)
    PGN_ELECTRIC_DRIVE_INFORMATION : UDINT := UDINT#16#1F206; (* < 127494 - Electric Drive Information *)
    PGN_ELECTRIC_ENERGY_STORAGE_INFORMATION : UDINT := UDINT#16#1F207; (* < 127495 - Electric Energy Storage Information *)
    PGN_TRIP_PARAMETERS_VESSEL : UDINT := UDINT#16#1F208; (* < 127496 - Trip Parameters, Vessel *)
    PGN_TRIP_PARAMETERS_ENGINE : UDINT := UDINT#16#1F209; (* < 127497 - Trip Parameters, Small Craft *)
    PGN_ENGINE_PARAMETERS_STATIC : UDINT := UDINT#16#1F20A; (* < 127498 - Engine Parameters, Static *)
    PGN_LOAD_CONTROLLER_CONNECTION_STATE_CONTROL : UDINT := UDINT#16#1F20C; (* < 127500 - Load Controller Connection State / Control *)
    PGN_BINARY_SWITCH_BANK_STATUS : UDINT := UDINT#16#1F20D; (* < 127501 - Binary Switch Bank Status *)
    PGN_SWITCH_BANK_CONTROL : UDINT := UDINT#16#1F20E; (* < 127502 - Switch Bank Control *)
    PGN_AC_INPUT_STATUS : UDINT := UDINT#16#1F20F; (* < 127503 - AC Input Status *)
    PGN_AC_OUTPUT_STATUS : UDINT := UDINT#16#1F210; (* < 127504 - AC Output Status *)
    PGN_FLUID_LEVEL : UDINT := UDINT#16#1F211; (* < 127505 - Fluid Level *)
    PGN_DCDETAILED_STATUS : UDINT := UDINT#16#1F212; (* < 127506 - DC Detailed Status *)
    PGN_CHARGER_STATUS : UDINT := UDINT#16#1F213; (* < 127507 - Charger Status *)
    PGN_BATTERY_STATUS : UDINT := UDINT#16#1F214; (* < 127508 - Battery Status *)
    PGN_INVERTER_STATUS : UDINT := UDINT#16#1F215; (* < 127509 - Inverter Status *)
    PGN_CHARGER_CONFIG_STATUS : UDINT := UDINT#16#1F216; (* < 127510 - Charger Configuration Status *)
    PGN_WATER_DEPTH : UDINT := UDINT#16#1F216; (* < 127510 - Charger Configuration Status *)
    PGN_INVERTER_CONFIG_STATUS : UDINT := UDINT#16#1F217; (* < 127511 - Inverter Configuration Status *)
    PGN_AGS_CONFIG_STATUS : UDINT := UDINT#16#1F218; (* < 127512 - AGS Configuration Status *)
    PGN_BATTERY_CONFIG_STATUS : UDINT := UDINT#16#1F219; (* < 127513 - Battery Configuration Status *)
    PGN_AGS_STATUS : UDINT := UDINT#16#1F21A; (* < 127514 - AGS Status *)
    PGN_AC_POWER_CURRENT_PHASE_A : UDINT := UDINT#16#1F300; (* < 127744 - AC Power / Current - Phase A *)
    PGN_AC_POWER_CURRENT_PHASE_B : UDINT := UDINT#16#1F301; (* < 127745 - AC Power / Current - Phase B *)
    PGN_AC_POWER_CURRENT_PHASE_C : UDINT := UDINT#16#1F302; (* < 127746 - AC Power / Current - Phase C *)
    PGN_AC_VOLTAGE_FREQUENCY_PHASE_A : UDINT := UDINT#16#1F303; (* < 127747 - AC Voltage / Frequency - Phase A *)
    PGN_AC_VOLTAGE_FREQUENCY_PHASE_B : UDINT := UDINT#16#1F304; (* < 127748 - AC Voltage / Frequency - Phase B *)
    PGN_AC_VOLTAGE_FREQUENCY_PHASE_C : UDINT := UDINT#16#1F305; (* < 127749 - AC Voltage / Frequency-Phase C *)
    PGN_CONVERTER_INVERTER_CHARGER_STATUS : UDINT := UDINT#16#1F306; (* < 127750 - Converter (Inverter/Charger) Status *)
    PGN_DC_VOLTAGE_CURRENT : UDINT := UDINT#16#1F307; (* < 127751 - DC Voltage / Current *)
    PGN_NAUTICAL_LEEWAY_ANGLE : UDINT := UDINT#16#1F400; (* < 128000 - Nautical Leeway Angle *)
    PGN_VESSEL_ACCELERATION : UDINT := UDINT#16#1F401; (* < 128001 - Vessel Acceleration *)
    PGN_ELECTRIC_DRIVE_STATUS_RAPID_UPDATE : UDINT := UDINT#16#1F402; (* < 128002 - Electric Drive Status, Rapid Update *)
    PGN_ELECTRIC_ENERGY_STORAGE_STATUS_RAPID_UPDATE : UDINT := UDINT#16#1F403; (* < 128003 - Electric Energy Storage Status, Rapid Update *)
    PGN_THRUSTER_CONTROL_STATUS : UDINT := UDINT#16#1F406; (* < 128006 - Thruster Control Status *)
    PGN_THRUSTER_INFORMATION : UDINT := UDINT#16#1F407; (* < 128007 - Thruster Information *)
    PGN_THRUSTER_MOTOR_STATUS : UDINT := UDINT#16#1F408; (* < 128008 - Thruster Motor Status *)
    PGN_SPEED_WATERREF : UDINT := UDINT#16#1F503; (* < 128259 - Speed *)
    PGN_WATER_DEPTH_128267 : UDINT := UDINT#16#1F50B; (* < 128267 - Water Depth *)
    PGN_DISTANCED_LOG : UDINT := UDINT#16#1F513; (* < 128275 - Distance Log *)
    PGN_TRACKED_TARGET_DATA : UDINT := UDINT#16#1F608; (* < 128520 - Tracked Target Data *)
    PGN_ELEVATOR_CAR_STATUS : UDINT := UDINT#16#1F61A; (* < 128538 - Elevator Car Status *)
    PGN_ELEVATOR_MOTOR_CONTROL : UDINT := UDINT#16#1F700; (* < 128768 - Elevator Motor Control *)
    PGN_ELEVATOR_DECK_PUSH_BUTTON : UDINT := UDINT#16#1F701; (* < 128769 - Elevator Deck Push Button *)
    PGN_WINDLASS_CONTROL_STATUS : UDINT := UDINT#16#1F708; (* < 128776 - Windlass Control Status *)
    PGN_ANCHOR_WINDLASS_OPERATING_STATUS : UDINT := UDINT#16#1F709; (* < 128777 - Anchor Windlass Operating Status *)
    PGN_ANCHOR_WINDLASS_MONITORING_STATUS : UDINT := UDINT#16#1F70A; (* < 128778 - Anchor Windlass Monitoring Status *)
    PGN_LINEAR_ACTUATOR_CONTROL_STATUS : UDINT := UDINT#16#1F70C; (* < 128780 - Linear Actuator Control/Status *)
    PGN_POSITION_RAPID_UPDATE : UDINT := UDINT#16#1F801; (* < 129025 - Position, Rapid Update *)
    PGN_COG_SOG_RAPID_UPDATE : UDINT := UDINT#16#1F802; (* < 129026 - COG & SOG, Rapid Update *)
    PGN_POSITION_DELTA_HP_RAPID_UPD : UDINT := UDINT#16#1F803; (* < 129027 - Position Delta, High Precision Rapid Update *)
    PGN_ALTITUDE_DELTA_HP_RAPID_UPD : UDINT := UDINT#16#1F804; (* < 129028 - Altitude Delta, High Precision Rapid Update *)
    PGN_GNSS_POSITION_DATA : UDINT := UDINT#16#1F805; (* < 129029 - GNSS Position Data *)
    PGN_NMEA_TIME_DATE : UDINT := UDINT#16#1F809; (* < 129033 - Time & Date *)
    PGN_AIS_CLASSA_POSITION_REPORT : UDINT := UDINT#16#1F80E; (* < 129038 - AIS Class A Position Report *)
    PGN_AIS_CLASSB_POSITION_REPORT : UDINT := UDINT#16#1F80F; (* < 129039 - AIS Class B Position Report *)
    PGN_AIS_CLASSB_EXTPOS_REPORT : UDINT := UDINT#16#1F810; (* < 129040 - AIS Class B Extended Position Report *)
    PGN_AIS_AIDS_TO_NAVIGATION_ATON_REPORT : UDINT := UDINT#16#1F811; (* < 129041 - AIS Aids to Navigation (AtoN) Report *)
    PGN_DATUM : UDINT := UDINT#16#1F814; (* < 129044 - Datum *)
    PGN_USER_DATUM_SETTINGS : UDINT := UDINT#16#1F815; (* < 129045 - User Datum Settings *)
    PGN_CROSS_TRACK_ERROR : UDINT := UDINT#16#1F903; (* < 129283 - Cross Track Error *)
    PGN_NAVIGATION_DATA : UDINT := UDINT#16#1F904; (* < 129284 - Navigation Data *)
    PGN_NAVIGATION_ROUTEWP_INFO : UDINT := UDINT#16#1F905; (* < 129285 - Navigation - Route/WP information *)
    PGN_SET_DRIFT_RAPID_UPDATE : UDINT := UDINT#16#1F90B; (* < 129291 - Set & Drift, Rapid Update *)
    PGN_TIME_TOFROM_MARK : UDINT := UDINT#16#1F915; (* < 129301 - Time to/from Mark *)
    PGN_BEARING_DIST_BET_TWO_MARKS : UDINT := UDINT#16#1F916; (* < 129302 - Bearing and Distance between two Marks *)
    PGN_GNSS_CONTROL_STATUS : UDINT := UDINT#16#1FA02; (* < 129538 - GNSS Control Status *)
    PGN_GNSS_DOPS : UDINT := UDINT#16#1FA03; (* < 129539 - GNSS DOPs *)
    PGN_GNSS_SATS_IN_VIEW : UDINT := UDINT#16#1FA04; (* < 129540 - GNSS Sats in View *)
    PGN_ALMANAC_DATA : UDINT := UDINT#16#1FA05; (* < 129541 - GPS Almanac Data *)
    PGN_GNSS_PSEUDOOR_NOISE_STATIST : UDINT := UDINT#16#1FA06; (* < 129542 - GNSS Pseudorange Noise Statistics *)
    PGN_GNSS_RAIM_OUTPUT : UDINT := UDINT#16#1FA09; (* < 129545 - GNSS RAIM Output *)
    PGN_GNSS_RAIM_SETTINGS : UDINT := UDINT#16#1FA0A; (* < 129546 - GNSS RAIM Settings *)
    PGN_GNSS_PSEUDOOR_ERROR_STATIST : UDINT := UDINT#16#1FA0B; (* < 129547 - GNSS Pseudorange Error Statistics *)
    PGN_DGNSS_CORRECTIONS : UDINT := UDINT#16#1FA0D; (* < 129549 - DGNSS Corrections *)
    PGN_GNSS_DIFF_CORR_RECEI_INTERF : UDINT := UDINT#16#1FA0E; (* < 129550 - GNSS Differential Correction Receiver Interface *)
    PGN_GNSS_DIFF_CORR_RECEIVE_SIGN : UDINT := UDINT#16#1FA0F; (* < 129551 - GNSS Differential Correction Receiver Signal *)
    PGN_GLONASS_ALMANAC_DATA : UDINT := UDINT#16#1FA14; (* < 129556 - GLONASS Almanac Data *)
    PGN_AIS_DGNSS_BROADC_BIN_MESSAG : UDINT := UDINT#16#1FB00; (* < 129792 - AIS DGNSS Broadcast Binary Message *)
    PGN_AIS_UTC_AND_DATE_REPORT : UDINT := UDINT#16#1FB01; (* < 129793 - AIS UTC and Date Report *)
    PGN_AIS_CLASS_A_STAT_VOYAGE_DAT : UDINT := UDINT#16#1FB02; (* < 129794 - AIS Class A Static and Voyage Related Data *)
    PGN_AIS_ADDRESSED_BINARY_MESSAG : UDINT := UDINT#16#1FB03; (* < 129795 - AIS Addressed Binary Message *)
    PGN_AIS_ACKNOWLEDGE : UDINT := UDINT#16#1FB04; (* < 129796 - AIS Acknowledge *)
    PGN_AIS_BINARY_BROADCAST_MESSAG : UDINT := UDINT#16#1FB05; (* < 129797 - AIS Binary Broadcast Message *)
    PGN_AIS_SAR_AIRCRAFT_POS_REPORT : UDINT := UDINT#16#1FB06; (* < 129798 - AIS SAR Aircraft Position Report *)
    PGN_RADIO_FREQUENCY_MODE_POWER : UDINT := UDINT#16#1FB07; (* < 129799 - Radio Frequency/Mode/Power *)
    PGN_AIS_UTC_DATE_INQUIRY : UDINT := UDINT#16#1FB08; (* < 129800 - AIS UTC/Date Inquiry *)
    PGN_AIS_ADDRESS_SAFE_REL_MESSAG : UDINT := UDINT#16#1FB09; (* < 129801 - AIS Addressed Safety Related Message *)
    PGN_AIS_SAFE_RELD_BROADC_MESSAG : UDINT := UDINT#16#1FB0A; (* < 129802 - AIS Safety Related Broadcast Message *)
    PGN_AIS_INTERROGATION : UDINT := UDINT#16#1FB0B; (* < 129803 - AIS Interrogation *)
    PGN_AIS_ASSIGNMENT_MODE_COMMAND : UDINT := UDINT#16#1FB0C; (* < 129804 - AIS Assignment Mode Command *)
    PGN_AIS_DATA_LINK_MANAGEMENT_MESSAGE : UDINT := UDINT#16#1FB0D; (* < 129805 - AIS Data Link Management Message *)
    PGN_AIS_CHANNEL_MANAGEMENT : UDINT := UDINT#16#1FB0E; (* < 129806 - AIS Channel Management *)
    PGN_AIS_CLASS_B_GROUP_ASSIGNMENT : UDINT := UDINT#16#1FB0F; (* < 129807 - AIS Class B Group Assignment *)
    PGN_DSC_CALL_INFORMATION : UDINT := UDINT#16#1FB10; (* < 129808 - DSC Call Information *)
    PGN_AIS_CLASS_B_CS_STATIC_DATA_REPORT_PART_A : UDINT := UDINT#16#1FB11; (* < 129809 - AIS Class B "CS" Static Data Report, Part A *)
    PGN_AIS_CLASS_B_CS_STATIC_DATA_REPORT_PART_B : UDINT := UDINT#16#1FB12; (* < 129810 - AIS Class B "CS" Static Data Report, Part B *)
    PGN_AIS_SINGLE_SLOT_BINARY_MESSAGE_DEPRECATED : UDINT := UDINT#16#1FB13; (* < 129811 - AIS Single Slot Binary Message - DEPRECATED *)
    PGN_AIS_MULTI_SLOT_BINARY_MESSAGE_DEPRECATED : UDINT := UDINT#16#1FB14; (* < 129812 - AIS Multi Slot Binary Message - DEPRECATED *)
    PGN_AIS_LONG_RANGE_BROADCAST_MESSAGE : UDINT := UDINT#16#1FB15; (* < 129813 - AIS Long-Range Broadcast Message *)
    PGN_AIS_SINGLE_SLOT_BINARY_MESSAGE : UDINT := UDINT#16#1FB16; (* < 129814 - AIS Single Slot Binary Message *)
    PGN_AIS_MULTI_SLOT_BINARY_MESSAGE : UDINT := UDINT#16#1FB17; (* < 129815 - AIS Multi Slot Binary Message *)
    PGN_AIS_ACKNOWLEDGE_129816 : UDINT := UDINT#16#1FB18; (* < 129816 - AIS Acknowledge *)
    PGN_LORAN_C_TD_DATA : UDINT := UDINT#16#1FC04; (* < 130052 - Loran-C TD Data *)
    PGN_LORAN_C_RANGE_DATA : UDINT := UDINT#16#1FC05; (* < 130053 - Loran-C Range Data *)
    PGN_LORAN_C_SIGNAL_DATA : UDINT := UDINT#16#1FC06; (* < 130054 - Loran-C Signal Data *)
    PGN_LABEL : UDINT := UDINT#16#1FC0C; (* < 130060 - Label *)
    PGN_CHANNEL_SOURCE_CONFIGURATION : UDINT := UDINT#16#1FC0D; (* < 130061 - Channel Source Configuration *)
    PGN_ROUTE_WP_SERVICE_DB_LIST : UDINT := UDINT#16#1FC10; (* < 130064 - Route and WP Service - Database List *)
    PGN_ROUTE_WP_SERVICE_ROUTE_LIST : UDINT := UDINT#16#1FC11; (* < 130065 - Route and WP Service - Route List *)
    PGN_ROUTE_WP_SERVICE_WP_ATTRIB : UDINT := UDINT#16#1FC12; (* < 130066 - Route and WP Service - Route/WP-List Attributes *)
    PGN_ROUTE_WP_SERVICE_WP_NAM_POS : UDINT := UDINT#16#1FC13; (* < 130067 - Route and WP Service - Route - WP Name & Position *)
    PGN_ROUTE_WP_SERVICE_QP_NAME : UDINT := UDINT#16#1FC14; (* < 130068 - Route and WP Service - Route - WP Name *)
    PGN_ROUTE_WP_SERVICE_XTE_LIMIT : UDINT := UDINT#16#1FC15; (* < 130069 - Route and WP Service - XTE Limit & Navigation Method *)
    PGN_ROUTE_WP_SERVICE_WP_COMMENT : UDINT := UDINT#16#1FC16; (* < 130070 - Route and WP Service - WP Comment *)
    PGN_ROUTE_WP_SERVICE_ROUTE_COM : UDINT := UDINT#16#1FC17; (* < 130071 - Route and WP Service - Route Comment *)
    PGN_ROUTE_WP_SERVICE_DB_COMMENT : UDINT := UDINT#16#1FC18; (* < 130072 - Route and WP Service - Database Comment *)
    PGN_ROUTE_WP_SERVICE_RADIU_TURN : UDINT := UDINT#16#1FC19; (* < 130073 - Route and WP Service - Radius of Turn *)
    PGN_ROUTE_WP_SERVICE_WP_LIS_NAM : UDINT := UDINT#16#1FC1A; (* < 130074 - Route and WP Service - WP List - WP Name & Position *)
    PGN_WIND_DATA : UDINT := UDINT#16#1FD02; (* < 130306 - Wind Data *)
    PGN_ENVIRONMENT_PARAMETERS : UDINT := UDINT#16#1FD06; (* < 130310 - Environmental Parameters *)
    PGN_ENVIRONMENT_PARAMETERS_2 : UDINT := UDINT#16#1FD07; (* < 130311 - Environmental Parameters *)
    PGN_TEMPERATURE : UDINT := UDINT#16#1FD08; (* < 130312 - Temperature *)
    PGN_HUMIDITY : UDINT := UDINT#16#1FD09; (* < 130313 - Humidity *)
    PGN_ACTUAL_PRESSURE : UDINT := UDINT#16#1FD0A; (* < 130314 - Actual Pressure *)
    PGN_SET_PRESSURE : UDINT := UDINT#16#1FD0B; (* < 130315 - Set Pressure *)
    PGN_TEMPERATURE_EXTENDED_RANGE : UDINT := UDINT#16#1FD0C; (* < 130316 - Temperature- Extended Range *)
    PGN_TIDE_STATION_DATA : UDINT := UDINT#16#1FD10; (* < 130320 - Tide Station Data *)
    PGN_SALINITY_STATION_DATA : UDINT := UDINT#16#1FD11; (* < 130321 - Salinity Station Data *)
    PGN_CURRENT_STATION_DATA : UDINT := UDINT#16#1FD12; (* < 130322 - Current Station Data *)
    PGN_METEOROLOGICAL_STATION_DATA : UDINT := UDINT#16#1FD13; (* < 130323 - Meteorological Station Data *)
    PGN_MOORED_BUOY_STATION_DATA : UDINT := UDINT#16#1FD14; (* < 130324 - Moored Buoy Station Data *)
    PGN_LIGHTING_SYSTEM_SETTINGS : UDINT := UDINT#16#1FD1A; (* < 130330 - Lighting System Settings *)
    PGN_PAYLOAD_MASS : UDINT := UDINT#16#1FE00; (* < 130560 - Payload Mass *)
    PGN_LIGHTING_ZONE : UDINT := UDINT#16#1FE01; (* < 130561 - Lighting Zone *)
    PGN_LIGHTING_SCENE : UDINT := UDINT#16#1FE02; (* < 130562 - Lighting Scene *)
    PGN_LIGHTING_DEVICE : UDINT := UDINT#16#1FE03; (* < 130563 - Lighting Device *)
    PGN_LIGHTING_DEVICE_ENUMERATION : UDINT := UDINT#16#1FE04; (* < 130564 - Lighting Device Enumeration *)
    PGN_LIGHTING_COLOR_SEQUENCE : UDINT := UDINT#16#1FE05; (* < 130565 - Lighting Color Sequence *)
    PGN_LIGHTING_PROGRAM : UDINT := UDINT#16#1FE06; (* < 130566 - Lighting Program *)
    PGN_WATERMAKER_INPUT_SETTING_AND_STATUS : UDINT := UDINT#16#1FE07; (* < 130567 - Watermaker Input Setting and Status *)
    PGN_ENTERTAINMENT_DIAGNOSTIC_STATUS : UDINT := UDINT#16#1FE08; (* < 130568 - Entertainment - Diagnostic Status *)
    PGN_ENTERTAINMENT_CURRENT_FILE_AND_STATUS : UDINT := UDINT#16#1FE09; (* < 130569 - Entertainment - Current File and Status *)
    PGN_ENTERTAINMENT_LIBRARY_DATA_FILE : UDINT := UDINT#16#1FE0A; (* < 130570 - Entertainment - Library Data File *)
    PGN_ENTERTAINMENT_LIBRARY_DATA_GROUP : UDINT := UDINT#16#1FE0B; (* < 130571 - Entertainment - Library Data Group *)
    PGN_ENTERTAINMENT_LIBRARY_DATA_SEARCH : UDINT := UDINT#16#1FE0C; (* < 130572 - Entertainment - Library Data Search *)
    PGN_ENTERTAINMENT_SUPPORTED_SOURCE_DATA : UDINT := UDINT#16#1FE0D; (* < 130573 - Entertainment - Supported Source Data *)
    PGN_ENTERTAINMENT_SUPPORTED_ZONE_DATA : UDINT := UDINT#16#1FE0E; (* < 130574 - Entertainment - Supported Zone Data *)
    PGN_ENTERTAINMENT_PARENTAL_CONTROL_STATUS : UDINT := UDINT#16#1FE0F; (* < 130575 - Entertainment - Parental Control Status *)
    PGN_SMALL_CRAFT_STATUS : UDINT := UDINT#16#1FE10; (* < 130576 - Small Craft Status *)
    PGN_DIRECTION_DATA : UDINT := UDINT#16#1FE11; (* < 130577 - Direction Data *)
    PGN_VESSEL_SPEED_COMPONENTS : UDINT := UDINT#16#1FE12; (* < 130578 - Vessel Speed Components *)
    PGN_ENTERTAINMENT_SYSTEM_CONFIGURATION : UDINT := UDINT#16#1FE13; (* < 130579 - Entertainment - System Configuration *)
    PGN_ENTERTAINMENT_SYSTEM_CONFIGURATION_STATUS : UDINT := UDINT#16#1FE14; (* < 130580 - Entertainment - System Configuration Status *)
    PGN_ENTERTAINMENT_ZONE_CONFIGURATION_STATUS_DEPRECATED : UDINT := UDINT#16#1FE15; (* < 130581 - Entertainment - Zone Configuration Status - DEPRECATED *)
    PGN_ENTERTAINMENT_ZONE_VOLUME : UDINT := UDINT#16#1FE16; (* < 130582 - Entertainment - Zone Volume *)
    PGN_ENTERTAINMENT_AVAILABLE_AUDIO_EQ_PRESETS : UDINT := UDINT#16#1FE17; (* < 130583 - Entertainment - Available Audio EQ Presets *)
    PGN_ENTERTAINMENT_BLUETOOTH_DEVICES : UDINT := UDINT#16#1FE18; (* < 130584 - Entertainment - Bluetooth Devices *)
    PGN_ENTERTAINMENT_BLUETOOTH_SOURCE_STATUS : UDINT := UDINT#16#1FE19; (* < 130585 - Entertainment - Bluetooth Source Status *)
    PGN_ENTERTAINMENT_ZONE_CONFIGURATION_STATUS : UDINT := UDINT#16#1FE1A; (* < 130586 - Entertainment - Zone Configuration Status *)
    PGN_PROPRIETARY_B_PAGE_1_FIRST_ENTRY : UDINT := UDINT#16#1FF00; (* < 130816 - PropB1_00 *)
    PGN_PROPRIETARY_B_PAGE_1 : UDINT := UDINT#16#1FF01; (* < 130817 - PropB1_01 *)
    PGN_PROPRIETARY_B_PAGE_1_130818 : UDINT := UDINT#16#1FF02; (* < 130818 - PropB1_02 *)
    PGN_PROPRIETARY_B_PAGE_1_130819 : UDINT := UDINT#16#1FF03; (* < 130819 - PropB1_03 *)
    PGN_PROPRIETARY_B_PAGE_1_130820 : UDINT := UDINT#16#1FF04; (* < 130820 - PropB1_04 *)
    PGN_PROPRIETARY_B_PAGE_1_130821 : UDINT := UDINT#16#1FF05; (* < 130821 - PropB1_05 *)
    PGN_PROPRIETARY_B_PAGE_1_130822 : UDINT := UDINT#16#1FF06; (* < 130822 - PropB1_06 *)
    PGN_PROPRIETARY_B_PAGE_1_130823 : UDINT := UDINT#16#1FF07; (* < 130823 - PropB1_07 *)
    PGN_PROPRIETARY_B_PAGE_1_130824 : UDINT := UDINT#16#1FF08; (* < 130824 - PropB1_08 *)
    PGN_PROPRIETARY_B_PAGE_1_130825 : UDINT := UDINT#16#1FF09; (* < 130825 - PropB1_09 *)
    PGN_PROPRIETARY_B_PAGE_1_130826 : UDINT := UDINT#16#1FF0A; (* < 130826 - PropB1_0A *)
    PGN_PROPRIETARY_B_PAGE_1_130827 : UDINT := UDINT#16#1FF0B; (* < 130827 - PropB1_0B *)
    PGN_PROPRIETARY_B_PAGE_1_130828 : UDINT := UDINT#16#1FF0C; (* < 130828 - PropB1_0C *)
    PGN_PROPRIETARY_B_PAGE_1_130829 : UDINT := UDINT#16#1FF0D; (* < 130829 - PropB1_0D *)
    PGN_PROPRIETARY_B_PAGE_1_130830 : UDINT := UDINT#16#1FF0E; (* < 130830 - PropB1_0E *)
    PGN_PROPRIETARY_B_PAGE_1_130831 : UDINT := UDINT#16#1FF0F; (* < 130831 - PropB1_0F *)
    PGN_PROPRIETARY_B_PAGE_1_130832 : UDINT := UDINT#16#1FF10; (* < 130832 - PropB1_10 *)
    PGN_PROPRIETARY_B_PAGE_1_130833 : UDINT := UDINT#16#1FF11; (* < 130833 - PropB1_11 *)
    PGN_PROPRIETARY_B_PAGE_1_130834 : UDINT := UDINT#16#1FF12; (* < 130834 - PropB1_12 *)
    PGN_PROPRIETARY_B_PAGE_1_130835 : UDINT := UDINT#16#1FF13; (* < 130835 - PropB1_13 *)
    PGN_PROPRIETARY_B_PAGE_1_130836 : UDINT := UDINT#16#1FF14; (* < 130836 - PropB1_14 *)
    PGN_PROPRIETARY_B_PAGE_1_130837 : UDINT := UDINT#16#1FF15; (* < 130837 - PropB1_15 *)
    PGN_PROPRIETARY_B_PAGE_1_130838 : UDINT := UDINT#16#1FF16; (* < 130838 - PropB1_16 *)
    PGN_PROPRIETARY_B_PAGE_1_130839 : UDINT := UDINT#16#1FF17; (* < 130839 - PropB1_17 *)
    PGN_PROPRIETARY_B_PAGE_1_130840 : UDINT := UDINT#16#1FF18; (* < 130840 - PropB1_18 *)
    PGN_PROPRIETARY_B_PAGE_1_130841 : UDINT := UDINT#16#1FF19; (* < 130841 - PropB1_19 *)
    PGN_PROPRIETARY_B_PAGE_1_130842 : UDINT := UDINT#16#1FF1A; (* < 130842 - PropB1_1A *)
    PGN_PROPRIETARY_B_PAGE_1_130843 : UDINT := UDINT#16#1FF1B; (* < 130843 - PropB1_1B *)
    PGN_PROPRIETARY_B_PAGE_1_130844 : UDINT := UDINT#16#1FF1C; (* < 130844 - PropB1_1C *)
    PGN_PROPRIETARY_B_PAGE_1_130845 : UDINT := UDINT#16#1FF1D; (* < 130845 - PropB1_1D *)
    PGN_PROPRIETARY_B_PAGE_1_130846 : UDINT := UDINT#16#1FF1E; (* < 130846 - PropB1_1E *)
    PGN_PROPRIETARY_B_PAGE_1_130847 : UDINT := UDINT#16#1FF1F; (* < 130847 - PropB1_1F *)
    PGN_PROPRIETARY_B_PAGE_1_130848 : UDINT := UDINT#16#1FF20; (* < 130848 - PropB1_20 *)
    PGN_PROPRIETARY_B_PAGE_1_130849 : UDINT := UDINT#16#1FF21; (* < 130849 - PropB1_21 *)
    PGN_PROPRIETARY_B_PAGE_1_130850 : UDINT := UDINT#16#1FF22; (* < 130850 - PropB1_22 *)
    PGN_PROPRIETARY_B_PAGE_1_130851 : UDINT := UDINT#16#1FF23; (* < 130851 - PropB1_23 *)
    PGN_PROPRIETARY_B_PAGE_1_130852 : UDINT := UDINT#16#1FF24; (* < 130852 - PropB1_24 *)
    PGN_PROPRIETARY_B_PAGE_1_130853 : UDINT := UDINT#16#1FF25; (* < 130853 - PropB1_25 *)
    PGN_PROPRIETARY_B_PAGE_1_130854 : UDINT := UDINT#16#1FF26; (* < 130854 - PropB1_26 *)
    PGN_PROPRIETARY_B_PAGE_1_130855 : UDINT := UDINT#16#1FF27; (* < 130855 - PropB1_27 *)
    PGN_PROPRIETARY_B_PAGE_1_130856 : UDINT := UDINT#16#1FF28; (* < 130856 - PropB1_28 *)
    PGN_PROPRIETARY_B_PAGE_1_130857 : UDINT := UDINT#16#1FF29; (* < 130857 - PropB1_29 *)
    PGN_PROPRIETARY_B_PAGE_1_130858 : UDINT := UDINT#16#1FF2A; (* < 130858 - PropB1_2A *)
    PGN_PROPRIETARY_B_PAGE_1_130859 : UDINT := UDINT#16#1FF2B; (* < 130859 - PropB1_2B *)
    PGN_PROPRIETARY_B_PAGE_1_130860 : UDINT := UDINT#16#1FF2C; (* < 130860 - PropB1_2C *)
    PGN_PROPRIETARY_B_PAGE_1_130861 : UDINT := UDINT#16#1FF2D; (* < 130861 - PropB1_2D *)
    PGN_PROPRIETARY_B_PAGE_1_130862 : UDINT := UDINT#16#1FF2E; (* < 130862 - PropB1_2E *)
    PGN_PROPRIETARY_B_PAGE_1_130863 : UDINT := UDINT#16#1FF2F; (* < 130863 - PropB1_2F *)
    PGN_PROPRIETARY_B_PAGE_1_130864 : UDINT := UDINT#16#1FF30; (* < 130864 - PropB1_30 *)
    PGN_PROPRIETARY_B_PAGE_1_130865 : UDINT := UDINT#16#1FF31; (* < 130865 - PropB1_31 *)
    PGN_PROPRIETARY_B_PAGE_1_130866 : UDINT := UDINT#16#1FF32; (* < 130866 - PropB1_32 *)
    PGN_PROPRIETARY_B_PAGE_1_130867 : UDINT := UDINT#16#1FF33; (* < 130867 - PropB1_33 *)
    PGN_PROPRIETARY_B_PAGE_1_130868 : UDINT := UDINT#16#1FF34; (* < 130868 - PropB1_34 *)
    PGN_PROPRIETARY_B_PAGE_1_130869 : UDINT := UDINT#16#1FF35; (* < 130869 - PropB1_35 *)
    PGN_PROPRIETARY_B_PAGE_1_130870 : UDINT := UDINT#16#1FF36; (* < 130870 - PropB1_36 *)
    PGN_PROPRIETARY_B_PAGE_1_130871 : UDINT := UDINT#16#1FF37; (* < 130871 - PropB1_37 *)
    PGN_PROPRIETARY_B_PAGE_1_130872 : UDINT := UDINT#16#1FF38; (* < 130872 - PropB1_38 *)
    PGN_PROPRIETARY_B_PAGE_1_130873 : UDINT := UDINT#16#1FF39; (* < 130873 - PropB1_39 *)
    PGN_PROPRIETARY_B_PAGE_1_130874 : UDINT := UDINT#16#1FF3A; (* < 130874 - PropB1_3A *)
    PGN_PROPRIETARY_B_PAGE_1_130875 : UDINT := UDINT#16#1FF3B; (* < 130875 - PropB1_3B *)
    PGN_PROPRIETARY_B_PAGE_1_130876 : UDINT := UDINT#16#1FF3C; (* < 130876 - PropB1_3C *)
    PGN_PROPRIETARY_B_PAGE_1_130877 : UDINT := UDINT#16#1FF3D; (* < 130877 - PropB1_3D *)
    PGN_PROPRIETARY_B_PAGE_1_130878 : UDINT := UDINT#16#1FF3E; (* < 130878 - PropB1_3E *)
    PGN_PROPRIETARY_B_PAGE_1_130879 : UDINT := UDINT#16#1FF3F; (* < 130879 - PropB1_3F *)
    PGN_PROPRIETARY_B_PAGE_1_130880 : UDINT := UDINT#16#1FF40; (* < 130880 - PropB1_40 *)
    PGN_PROPRIETARY_B_PAGE_1_130881 : UDINT := UDINT#16#1FF41; (* < 130881 - PropB1_41 *)
    PGN_PROPRIETARY_B_PAGE_1_130882 : UDINT := UDINT#16#1FF42; (* < 130882 - PropB1_42 *)
    PGN_PROPRIETARY_B_PAGE_1_130883 : UDINT := UDINT#16#1FF43; (* < 130883 - PropB1_43 *)
    PGN_PROPRIETARY_B_PAGE_1_130884 : UDINT := UDINT#16#1FF44; (* < 130884 - PropB1_44 *)
    PGN_PROPRIETARY_B_PAGE_1_130885 : UDINT := UDINT#16#1FF45; (* < 130885 - PropB1_45 *)
    PGN_PROPRIETARY_B_PAGE_1_130886 : UDINT := UDINT#16#1FF46; (* < 130886 - PropB1_46 *)
    PGN_PROPRIETARY_B_PAGE_1_130887 : UDINT := UDINT#16#1FF47; (* < 130887 - PropB1_47 *)
    PGN_PROPRIETARY_B_PAGE_1_130888 : UDINT := UDINT#16#1FF48; (* < 130888 - PropB1_48 *)
    PGN_PROPRIETARY_B_PAGE_1_130889 : UDINT := UDINT#16#1FF49; (* < 130889 - PropB1_49 *)
    PGN_PROPRIETARY_B_PAGE_1_130890 : UDINT := UDINT#16#1FF4A; (* < 130890 - PropB1_4A *)
    PGN_PROPRIETARY_B_PAGE_1_130891 : UDINT := UDINT#16#1FF4B; (* < 130891 - PropB1_4B *)
    PGN_PROPRIETARY_B_PAGE_1_130892 : UDINT := UDINT#16#1FF4C; (* < 130892 - PropB1_4C *)
    PGN_PROPRIETARY_B_PAGE_1_130893 : UDINT := UDINT#16#1FF4D; (* < 130893 - PropB1_4D *)
    PGN_PROPRIETARY_B_PAGE_1_130894 : UDINT := UDINT#16#1FF4E; (* < 130894 - PropB1_4E *)
    PGN_PROPRIETARY_B_PAGE_1_130895 : UDINT := UDINT#16#1FF4F; (* < 130895 - PropB1_4F *)
    PGN_PROPRIETARY_B_PAGE_1_130896 : UDINT := UDINT#16#1FF50; (* < 130896 - PropB1_50 *)
    PGN_PROPRIETARY_B_PAGE_1_130897 : UDINT := UDINT#16#1FF51; (* < 130897 - PropB1_51 *)
    PGN_PROPRIETARY_B_PAGE_1_130898 : UDINT := UDINT#16#1FF52; (* < 130898 - PropB1_52 *)
    PGN_PROPRIETARY_B_PAGE_1_130899 : UDINT := UDINT#16#1FF53; (* < 130899 - PropB1_53 *)
    PGN_PROPRIETARY_B_PAGE_1_130900 : UDINT := UDINT#16#1FF54; (* < 130900 - PropB1_54 *)
    PGN_PROPRIETARY_B_PAGE_1_130901 : UDINT := UDINT#16#1FF55; (* < 130901 - PropB1_55 *)
    PGN_PROPRIETARY_B_PAGE_1_130902 : UDINT := UDINT#16#1FF56; (* < 130902 - PropB1_56 *)
    PGN_PROPRIETARY_B_PAGE_1_130903 : UDINT := UDINT#16#1FF57; (* < 130903 - PropB1_57 *)
    PGN_PROPRIETARY_B_PAGE_1_130904 : UDINT := UDINT#16#1FF58; (* < 130904 - PropB1_58 *)
    PGN_PROPRIETARY_B_PAGE_1_130905 : UDINT := UDINT#16#1FF59; (* < 130905 - PropB1_59 *)
    PGN_PROPRIETARY_B_PAGE_1_130906 : UDINT := UDINT#16#1FF5A; (* < 130906 - PropB1_5A *)
    PGN_PROPRIETARY_B_PAGE_1_130907 : UDINT := UDINT#16#1FF5B; (* < 130907 - PropB1_5B *)
    PGN_PROPRIETARY_B_PAGE_1_130908 : UDINT := UDINT#16#1FF5C; (* < 130908 - PropB1_5C *)
    PGN_PROPRIETARY_B_PAGE_1_130909 : UDINT := UDINT#16#1FF5D; (* < 130909 - PropB1_5D *)
    PGN_PROPRIETARY_B_PAGE_1_130910 : UDINT := UDINT#16#1FF5E; (* < 130910 - PropB1_5E *)
    PGN_PROPRIETARY_B_PAGE_1_130911 : UDINT := UDINT#16#1FF5F; (* < 130911 - PropB1_5F *)
    PGN_PROPRIETARY_B_PAGE_1_130912 : UDINT := UDINT#16#1FF60; (* < 130912 - PropB1_60 *)
    PGN_PROPRIETARY_B_PAGE_1_130913 : UDINT := UDINT#16#1FF61; (* < 130913 - PropB1_61 *)
    PGN_PROPRIETARY_B_PAGE_1_130914 : UDINT := UDINT#16#1FF62; (* < 130914 - PropB1_62 *)
    PGN_PROPRIETARY_B_PAGE_1_130915 : UDINT := UDINT#16#1FF63; (* < 130915 - PropB1_63 *)
    PGN_PROPRIETARY_B_PAGE_1_130916 : UDINT := UDINT#16#1FF64; (* < 130916 - PropB1_64 *)
    PGN_PROPRIETARY_B_PAGE_1_130917 : UDINT := UDINT#16#1FF65; (* < 130917 - PropB1_65 *)
    PGN_PROPRIETARY_B_PAGE_1_130918 : UDINT := UDINT#16#1FF66; (* < 130918 - PropB1_66 *)
    PGN_PROPRIETARY_B_PAGE_1_130919 : UDINT := UDINT#16#1FF67; (* < 130919 - PropB1_67 *)
    PGN_PROPRIETARY_B_PAGE_1_130920 : UDINT := UDINT#16#1FF68; (* < 130920 - PropB1_68 *)
    PGN_PROPRIETARY_B_PAGE_1_130921 : UDINT := UDINT#16#1FF69; (* < 130921 - PropB1_69 *)
    PGN_PROPRIETARY_B_PAGE_1_130922 : UDINT := UDINT#16#1FF6A; (* < 130922 - PropB1_6A *)
    PGN_PROPRIETARY_B_PAGE_1_130923 : UDINT := UDINT#16#1FF6B; (* < 130923 - PropB1_6B *)
    PGN_PROPRIETARY_B_PAGE_1_130924 : UDINT := UDINT#16#1FF6C; (* < 130924 - PropB1_6C *)
    PGN_PROPRIETARY_B_PAGE_1_130925 : UDINT := UDINT#16#1FF6D; (* < 130925 - PropB1_6D *)
    PGN_PROPRIETARY_B_PAGE_1_130926 : UDINT := UDINT#16#1FF6E; (* < 130926 - PropB1_6E *)
    PGN_PROPRIETARY_B_PAGE_1_130927 : UDINT := UDINT#16#1FF6F; (* < 130927 - PropB1_6F *)
    PGN_PROPRIETARY_B_PAGE_1_130928 : UDINT := UDINT#16#1FF70; (* < 130928 - PropB1_70 *)
    PGN_PROPRIETARY_B_PAGE_1_130929 : UDINT := UDINT#16#1FF71; (* < 130929 - PropB1_71 *)
    PGN_PROPRIETARY_B_PAGE_1_130930 : UDINT := UDINT#16#1FF72; (* < 130930 - PropB1_72 *)
    PGN_PROPRIETARY_B_PAGE_1_130931 : UDINT := UDINT#16#1FF73; (* < 130931 - PropB1_73 *)
    PGN_PROPRIETARY_B_PAGE_1_130932 : UDINT := UDINT#16#1FF74; (* < 130932 - PropB1_74 *)
    PGN_PROPRIETARY_B_PAGE_1_130933 : UDINT := UDINT#16#1FF75; (* < 130933 - PropB1_75 *)
    PGN_PROPRIETARY_B_PAGE_1_130934 : UDINT := UDINT#16#1FF76; (* < 130934 - PropB1_76 *)
    PGN_PROPRIETARY_B_PAGE_1_130935 : UDINT := UDINT#16#1FF77; (* < 130935 - PropB1_77 *)
    PGN_PROPRIETARY_B_PAGE_1_130936 : UDINT := UDINT#16#1FF78; (* < 130936 - PropB1_78 *)
    PGN_PROPRIETARY_B_PAGE_1_130937 : UDINT := UDINT#16#1FF79; (* < 130937 - PropB1_79 *)
    PGN_PROPRIETARY_B_PAGE_1_130938 : UDINT := UDINT#16#1FF7A; (* < 130938 - PropB1_7A *)
    PGN_PROPRIETARY_B_PAGE_1_130939 : UDINT := UDINT#16#1FF7B; (* < 130939 - PropB1_7B *)
    PGN_PROPRIETARY_B_PAGE_1_130940 : UDINT := UDINT#16#1FF7C; (* < 130940 - PropB1_7C *)
    PGN_PROPRIETARY_B_PAGE_1_130941 : UDINT := UDINT#16#1FF7D; (* < 130941 - PropB1_7D *)
    PGN_PROPRIETARY_B_PAGE_1_130942 : UDINT := UDINT#16#1FF7E; (* < 130942 - PropB1_7E *)
    PGN_PROPRIETARY_B_PAGE_1_130943 : UDINT := UDINT#16#1FF7F; (* < 130943 - PropB1_7F *)
    PGN_PROPRIETARY_B_PAGE_1_130944 : UDINT := UDINT#16#1FF80; (* < 130944 - PropB1_80 *)
    PGN_PROPRIETARY_B_PAGE_1_130945 : UDINT := UDINT#16#1FF81; (* < 130945 - PropB1_81 *)
    PGN_PROPRIETARY_B_PAGE_1_130946 : UDINT := UDINT#16#1FF82; (* < 130946 - PropB1_82 *)
    PGN_PROPRIETARY_B_PAGE_1_130947 : UDINT := UDINT#16#1FF83; (* < 130947 - PropB1_83 *)
    PGN_PROPRIETARY_B_PAGE_1_130948 : UDINT := UDINT#16#1FF84; (* < 130948 - PropB1_84 *)
    PGN_PROPRIETARY_B_PAGE_1_130949 : UDINT := UDINT#16#1FF85; (* < 130949 - PropB1_85 *)
    PGN_PROPRIETARY_B_PAGE_1_130950 : UDINT := UDINT#16#1FF86; (* < 130950 - PropB1_86 *)
    PGN_PROPRIETARY_B_PAGE_1_130951 : UDINT := UDINT#16#1FF87; (* < 130951 - PropB1_87 *)
    PGN_PROPRIETARY_B_PAGE_1_130952 : UDINT := UDINT#16#1FF88; (* < 130952 - PropB1_88 *)
    PGN_PROPRIETARY_B_PAGE_1_130953 : UDINT := UDINT#16#1FF89; (* < 130953 - PropB1_89 *)
    PGN_PROPRIETARY_B_PAGE_1_130954 : UDINT := UDINT#16#1FF8A; (* < 130954 - PropB1_8A *)
    PGN_PROPRIETARY_B_PAGE_1_130955 : UDINT := UDINT#16#1FF8B; (* < 130955 - PropB1_8B *)
    PGN_PROPRIETARY_B_PAGE_1_130956 : UDINT := UDINT#16#1FF8C; (* < 130956 - PropB1_8C *)
    PGN_PROPRIETARY_B_PAGE_1_130957 : UDINT := UDINT#16#1FF8D; (* < 130957 - PropB1_8D *)
    PGN_PROPRIETARY_B_PAGE_1_130958 : UDINT := UDINT#16#1FF8E; (* < 130958 - PropB1_8E *)
    PGN_PROPRIETARY_B_PAGE_1_130959 : UDINT := UDINT#16#1FF8F; (* < 130959 - PropB1_8F *)
    PGN_PROPRIETARY_B_PAGE_1_130960 : UDINT := UDINT#16#1FF90; (* < 130960 - PropB1_90 *)
    PGN_PROPRIETARY_B_PAGE_1_130961 : UDINT := UDINT#16#1FF91; (* < 130961 - PropB1_91 *)
    PGN_PROPRIETARY_B_PAGE_1_130962 : UDINT := UDINT#16#1FF92; (* < 130962 - PropB1_92 *)
    PGN_PROPRIETARY_B_PAGE_1_130963 : UDINT := UDINT#16#1FF93; (* < 130963 - PropB1_93 *)
    PGN_PROPRIETARY_B_PAGE_1_130964 : UDINT := UDINT#16#1FF94; (* < 130964 - PropB1_94 *)
    PGN_PROPRIETARY_B_PAGE_1_130965 : UDINT := UDINT#16#1FF95; (* < 130965 - PropB1_95 *)
    PGN_PROPRIETARY_B_PAGE_1_130966 : UDINT := UDINT#16#1FF96; (* < 130966 - PropB1_96 *)
    PGN_PROPRIETARY_B_PAGE_1_130967 : UDINT := UDINT#16#1FF97; (* < 130967 - PropB1_97 *)
    PGN_PROPRIETARY_B_PAGE_1_130968 : UDINT := UDINT#16#1FF98; (* < 130968 - PropB1_98 *)
    PGN_PROPRIETARY_B_PAGE_1_130969 : UDINT := UDINT#16#1FF99; (* < 130969 - PropB1_99 *)
    PGN_PROPRIETARY_B_PAGE_1_130970 : UDINT := UDINT#16#1FF9A; (* < 130970 - PropB1_9A *)
    PGN_PROPRIETARY_B_PAGE_1_130971 : UDINT := UDINT#16#1FF9B; (* < 130971 - PropB1_9B *)
    PGN_PROPRIETARY_B_PAGE_1_130972 : UDINT := UDINT#16#1FF9C; (* < 130972 - PropB1_9C *)
    PGN_PROPRIETARY_B_PAGE_1_130973 : UDINT := UDINT#16#1FF9D; (* < 130973 - PropB1_9D *)
    PGN_PROPRIETARY_B_PAGE_1_130974 : UDINT := UDINT#16#1FF9E; (* < 130974 - PropB1_9E *)
    PGN_PROPRIETARY_B_PAGE_1_130975 : UDINT := UDINT#16#1FF9F; (* < 130975 - PropB1_9F *)
    PGN_PROPRIETARY_B_PAGE_1_130976 : UDINT := UDINT#16#1FFA0; (* < 130976 - PropB1_A0 *)
    PGN_PROPRIETARY_B_PAGE_1_130977 : UDINT := UDINT#16#1FFA1; (* < 130977 - PropB1_A1 *)
    PGN_PROPRIETARY_B_PAGE_1_130978 : UDINT := UDINT#16#1FFA2; (* < 130978 - PropB1_A2 *)
    PGN_PROPRIETARY_B_PAGE_1_130979 : UDINT := UDINT#16#1FFA3; (* < 130979 - PropB1_A3 *)
    PGN_PROPRIETARY_B_PAGE_1_130980 : UDINT := UDINT#16#1FFA4; (* < 130980 - PropB1_A4 *)
    PGN_PROPRIETARY_B_PAGE_1_130981 : UDINT := UDINT#16#1FFA5; (* < 130981 - PropB1_A5 *)
    PGN_PROPRIETARY_B_PAGE_1_130982 : UDINT := UDINT#16#1FFA6; (* < 130982 - PropB1_A6 *)
    PGN_PROPRIETARY_B_PAGE_1_130983 : UDINT := UDINT#16#1FFA7; (* < 130983 - PropB1_A7 *)
    PGN_PROPRIETARY_B_PAGE_1_130984 : UDINT := UDINT#16#1FFA8; (* < 130984 - PropB1_A8 *)
    PGN_PROPRIETARY_B_PAGE_1_130985 : UDINT := UDINT#16#1FFA9; (* < 130985 - PropB1_A9 *)
    PGN_PROPRIETARY_B_PAGE_1_130986 : UDINT := UDINT#16#1FFAA; (* < 130986 - PropB1_AA *)
    PGN_PROPRIETARY_B_PAGE_1_130987 : UDINT := UDINT#16#1FFAB; (* < 130987 - PropB1_AB *)
    PGN_PROPRIETARY_B_PAGE_1_130988 : UDINT := UDINT#16#1FFAC; (* < 130988 - PropB1_AC *)
    PGN_PROPRIETARY_B_PAGE_1_130989 : UDINT := UDINT#16#1FFAD; (* < 130989 - PropB1_AD *)
    PGN_PROPRIETARY_B_PAGE_1_130990 : UDINT := UDINT#16#1FFAE; (* < 130990 - PropB1_AE *)
    PGN_PROPRIETARY_B_PAGE_1_130991 : UDINT := UDINT#16#1FFAF; (* < 130991 - PropB1_AF *)
    PGN_PROPRIETARY_B_PAGE_1_130992 : UDINT := UDINT#16#1FFB0; (* < 130992 - PropB1_B0 *)
    PGN_PROPRIETARY_B_PAGE_1_130993 : UDINT := UDINT#16#1FFB1; (* < 130993 - PropB1_B1 *)
    PGN_PROPRIETARY_B_PAGE_1_130994 : UDINT := UDINT#16#1FFB2; (* < 130994 - PropB1_B2 *)
    PGN_PROPRIETARY_B_PAGE_1_130995 : UDINT := UDINT#16#1FFB3; (* < 130995 - PropB1_B3 *)
    PGN_PROPRIETARY_B_PAGE_1_130996 : UDINT := UDINT#16#1FFB4; (* < 130996 - PropB1_B4 *)
    PGN_PROPRIETARY_B_PAGE_1_130997 : UDINT := UDINT#16#1FFB5; (* < 130997 - PropB1_B5 *)
    PGN_PROPRIETARY_B_PAGE_1_130998 : UDINT := UDINT#16#1FFB6; (* < 130998 - PropB1_B6 *)
    PGN_PROPRIETARY_B_PAGE_1_130999 : UDINT := UDINT#16#1FFB7; (* < 130999 - PropB1_B7 *)
    PGN_PROPRIETARY_B_PAGE_1_131000 : UDINT := UDINT#16#1FFB8; (* < 131000 - PropB1_B8 *)
    PGN_PROPRIETARY_B_PAGE_1_131001 : UDINT := UDINT#16#1FFB9; (* < 131001 - PropB1_B9 *)
    PGN_PROPRIETARY_B_PAGE_1_131002 : UDINT := UDINT#16#1FFBA; (* < 131002 - PropB1_BA *)
    PGN_PROPRIETARY_B_PAGE_1_131003 : UDINT := UDINT#16#1FFBB; (* < 131003 - PropB1_BB *)
    PGN_PROPRIETARY_B_PAGE_1_131004 : UDINT := UDINT#16#1FFBC; (* < 131004 - PropB1_BC *)
    PGN_PROPRIETARY_B_PAGE_1_131005 : UDINT := UDINT#16#1FFBD; (* < 131005 - PropB1_BD *)
    PGN_PROPRIETARY_B_PAGE_1_131006 : UDINT := UDINT#16#1FFBE; (* < 131006 - PropB1_BE *)
    PGN_PROPRIETARY_B_PAGE_1_131007 : UDINT := UDINT#16#1FFBF; (* < 131007 - PropB1_BF *)
    PGN_PROPRIETARY_B_PAGE_1_131008 : UDINT := UDINT#16#1FFC0; (* < 131008 - PropB1_C0 *)
    PGN_PROPRIETARY_B_PAGE_1_131009 : UDINT := UDINT#16#1FFC1; (* < 131009 - PropB1_C1 *)
    PGN_PROPRIETARY_B_PAGE_1_131010 : UDINT := UDINT#16#1FFC2; (* < 131010 - PropB1_C2 *)
    PGN_PROPRIETARY_B_PAGE_1_131011 : UDINT := UDINT#16#1FFC3; (* < 131011 - PropB1_C3 *)
    PGN_PROPRIETARY_B_PAGE_1_131012 : UDINT := UDINT#16#1FFC4; (* < 131012 - PropB1_C4 *)
    PGN_PROPRIETARY_B_PAGE_1_131013 : UDINT := UDINT#16#1FFC5; (* < 131013 - PropB1_C5 *)
    PGN_PROPRIETARY_B_PAGE_1_131014 : UDINT := UDINT#16#1FFC6; (* < 131014 - PropB1_C6 *)
    PGN_PROPRIETARY_B_PAGE_1_131015 : UDINT := UDINT#16#1FFC7; (* < 131015 - PropB1_C7 *)
    PGN_PROPRIETARY_B_PAGE_1_131016 : UDINT := UDINT#16#1FFC8; (* < 131016 - PropB1_C8 *)
    PGN_PROPRIETARY_B_PAGE_1_131017 : UDINT := UDINT#16#1FFC9; (* < 131017 - PropB1_C9 *)
    PGN_PROPRIETARY_B_PAGE_1_131018 : UDINT := UDINT#16#1FFCA; (* < 131018 - PropB1_CA *)
    PGN_PROPRIETARY_B_PAGE_1_131019 : UDINT := UDINT#16#1FFCB; (* < 131019 - PropB1_CB *)
    PGN_PROPRIETARY_B_PAGE_1_131020 : UDINT := UDINT#16#1FFCC; (* < 131020 - PropB1_CC *)
    PGN_PROPRIETARY_B_PAGE_1_131021 : UDINT := UDINT#16#1FFCD; (* < 131021 - PropB1_CD *)
    PGN_PROPRIETARY_B_PAGE_1_131022 : UDINT := UDINT#16#1FFCE; (* < 131022 - PropB1_CE *)
    PGN_PROPRIETARY_B_PAGE_1_131023 : UDINT := UDINT#16#1FFCF; (* < 131023 - PropB1_CF *)
    PGN_PROPRIETARY_B_PAGE_1_131024 : UDINT := UDINT#16#1FFD0; (* < 131024 - PropB1_D0 *)
    PGN_PROPRIETARY_B_PAGE_1_131025 : UDINT := UDINT#16#1FFD1; (* < 131025 - PropB1_D1 *)
    PGN_PROPRIETARY_B_PAGE_1_131026 : UDINT := UDINT#16#1FFD2; (* < 131026 - PropB1_D2 *)
    PGN_PROPRIETARY_B_PAGE_1_131027 : UDINT := UDINT#16#1FFD3; (* < 131027 - PropB1_D3 *)
    PGN_PROPRIETARY_B_PAGE_1_131028 : UDINT := UDINT#16#1FFD4; (* < 131028 - PropB1_D4 *)
    PGN_PROPRIETARY_B_PAGE_1_131029 : UDINT := UDINT#16#1FFD5; (* < 131029 - PropB1_D5 *)
    PGN_PROPRIETARY_B_PAGE_1_131030 : UDINT := UDINT#16#1FFD6; (* < 131030 - PropB1_D6 *)
    PGN_PROPRIETARY_B_PAGE_1_131031 : UDINT := UDINT#16#1FFD7; (* < 131031 - PropB1_D7 *)
    PGN_PROPRIETARY_B_PAGE_1_131032 : UDINT := UDINT#16#1FFD8; (* < 131032 - PropB1_D8 *)
    PGN_PROPRIETARY_B_PAGE_1_131033 : UDINT := UDINT#16#1FFD9; (* < 131033 - PropB1_D9 *)
    PGN_PROPRIETARY_B_PAGE_1_131034 : UDINT := UDINT#16#1FFDA; (* < 131034 - PropB1_DA *)
    PGN_PROPRIETARY_B_PAGE_1_131035 : UDINT := UDINT#16#1FFDB; (* < 131035 - PropB1_DB *)
    PGN_PROPRIETARY_B_PAGE_1_131036 : UDINT := UDINT#16#1FFDC; (* < 131036 - PropB1_DC *)
    PGN_PROPRIETARY_B_PAGE_1_131037 : UDINT := UDINT#16#1FFDD; (* < 131037 - PropB1_DD *)
    PGN_PROPRIETARY_B_PAGE_1_131038 : UDINT := UDINT#16#1FFDE; (* < 131038 - PropB1_DE *)
    PGN_PROPRIETARY_B_PAGE_1_131039 : UDINT := UDINT#16#1FFDF; (* < 131039 - PropB1_DF *)
    PGN_PROPRIETARY_B_PAGE_1_131040 : UDINT := UDINT#16#1FFE0; (* < 131040 - PropB1_E0 *)
    PGN_PROPRIETARY_B_PAGE_1_131041 : UDINT := UDINT#16#1FFE1; (* < 131041 - PropB1_E1 *)
    PGN_PROPRIETARY_B_PAGE_1_131042 : UDINT := UDINT#16#1FFE2; (* < 131042 - PropB1_E2 *)
    PGN_PROPRIETARY_B_PAGE_1_131043 : UDINT := UDINT#16#1FFE3; (* < 131043 - PropB1_E3 *)
    PGN_PROPRIETARY_B_PAGE_1_131044 : UDINT := UDINT#16#1FFE4; (* < 131044 - PropB1_E4 *)
    PGN_PROPRIETARY_B_PAGE_1_131045 : UDINT := UDINT#16#1FFE5; (* < 131045 - PropB1_E5 *)
    PGN_PROPRIETARY_B_PAGE_1_131046 : UDINT := UDINT#16#1FFE6; (* < 131046 - PropB1_E6 *)
    PGN_PROPRIETARY_B_PAGE_1_131047 : UDINT := UDINT#16#1FFE7; (* < 131047 - PropB1_E7 *)
    PGN_PROPRIETARY_B_PAGE_1_131048 : UDINT := UDINT#16#1FFE8; (* < 131048 - PropB1_E8 *)
    PGN_PROPRIETARY_B_PAGE_1_131049 : UDINT := UDINT#16#1FFE9; (* < 131049 - PropB1_E9 *)
    PGN_PROPRIETARY_B_PAGE_1_131050 : UDINT := UDINT#16#1FFEA; (* < 131050 - PropB1_EA *)
    PGN_PROPRIETARY_B_PAGE_1_131051 : UDINT := UDINT#16#1FFEB; (* < 131051 - PropB1_EB *)
    PGN_PROPRIETARY_B_PAGE_1_131052 : UDINT := UDINT#16#1FFEC; (* < 131052 - PropB1_EC *)
    PGN_PROPRIETARY_B_PAGE_1_131053 : UDINT := UDINT#16#1FFED; (* < 131053 - PropB1_ED *)
    PGN_PROPRIETARY_B_PAGE_1_131054 : UDINT := UDINT#16#1FFEE; (* < 131054 - PropB1_EE *)
    PGN_PROPRIETARY_B_PAGE_1_131055 : UDINT := UDINT#16#1FFEF; (* < 131055 - PropB1_EF *)
    PGN_PROPRIETARY_B_PAGE_1_131056 : UDINT := UDINT#16#1FFF0; (* < 131056 - PropB1_F0 *)
    PGN_PROPRIETARY_B_PAGE_1_131057 : UDINT := UDINT#16#1FFF1; (* < 131057 - PropB1_F1 *)
    PGN_PROPRIETARY_B_PAGE_1_131058 : UDINT := UDINT#16#1FFF2; (* < 131058 - PropB1_F2 *)
    PGN_PROPRIETARY_B_PAGE_1_131059 : UDINT := UDINT#16#1FFF3; (* < 131059 - PropB1_F3 *)
    PGN_PROPRIETARY_B_PAGE_1_131060 : UDINT := UDINT#16#1FFF4; (* < 131060 - PropB1_F4 *)
    PGN_PROPRIETARY_B_PAGE_1_131061 : UDINT := UDINT#16#1FFF5; (* < 131061 - PropB1_F5 *)
    PGN_PROPRIETARY_B_PAGE_1_131062 : UDINT := UDINT#16#1FFF6; (* < 131062 - PropB1_F6 *)
    PGN_PROPRIETARY_B_PAGE_1_131063 : UDINT := UDINT#16#1FFF7; (* < 131063 - PropB1_F7 *)
    PGN_PROPRIETARY_B_PAGE_1_131064 : UDINT := UDINT#16#1FFF8; (* < 131064 - PropB1_F8 *)
    PGN_PROPRIETARY_B_PAGE_1_131065 : UDINT := UDINT#16#1FFF9; (* < 131065 - PropB1_F9 *)
    PGN_PROPRIETARY_B_PAGE_1_131066 : UDINT := UDINT#16#1FFFA; (* < 131066 - PropB1_FA *)
    PGN_PROPRIETARY_B_PAGE_1_131067 : UDINT := UDINT#16#1FFFB; (* < 131067 - PropB1_FB *)
    PGN_PROPRIETARY_B_PAGE_1_131068 : UDINT := UDINT#16#1FFFC; (* < 131068 - PropB1_FC *)
    PGN_PROPRIETARY_B_PAGE_1_131069 : UDINT := UDINT#16#1FFFD; (* < 131069 - PropB1_FD *)
    PGN_PROPRIETARY_B_PAGE_1_131070 : UDINT := UDINT#16#1FFFE; (* < 131070 - PropB1_FE *)
    PGN_PROPRIETARY_B_PAGE_1_LAST_ENTRY : UDINT := UDINT#16#1FFFF; (* < 131071 - PropB1_FF *)
  END_VAR
END_GLOBALCONSTANTS
